C09104=1030.328,224.816,385.474,170.153,45.182,158.614
C09105=1030.334,225.065,385.447,170.156,45.180,158.614
C09106=1030.342,225.314,385.420,170.159,45.179,158.614
C09107=1030.349,225.562,385.392,170.162,45.178,158.614
C09108=1030.355,225.810,385.364,170.164,45.177,158.614
C09109=1030.361,226.059,385.337,170.167,45.176,158.614
C09110=1030.368,226.307,385.310,170.170,45.175,158.614
C09111=1030.375,226.555,385.283,170.173,45.174,158.614
C09112=1030.382,226.804,385.255,170.176,45.173,158.614
C09113=1030.388,227.052,385.227,170.180,45.172,158.614
C09114=1030.395,227.301,385.200,170.183,45.171,158.614
C09115=1030.402,227.549,385.173,170.186,45.170,158.614
C09116=1030.409,227.798,385.145,170.189,45.169,158.614
C09117=1030.416,228.046,385.118,170.192,45.168,158.615
C09118=1030.422,228.294,385.090,170.195,45.167,158.615
C09119=1030.428,228.543,385.062,170.198,45.166,158.615
C09120=1030.435,228.791,385.035,170.200,45.165,158.615
C09121=1030.442,229.039,385.007,170.203,45.164,158.615
C09122=1030.448,229.288,384.979,170.206,45.163,158.615
C09123=1030.455,229.536,384.952,170.209,45.162,158.615
C09124=1030.462,229.785,384.924,170.212,45.161,158.615
C09125=1030.468,230.033,384.896,170.215,45.160,158.615
C09126=1030.475,230.282,384.868,170.219,45.159,158.615
C09127=1030.482,230.530,384.841,170.222,45.158,158.616
C09128=1030.488,230.779,384.813,170.225,45.157,158.616
C09129=1030.495,231.027,384.785,170.228,45.157,158.616
C09130=1030.501,231.275,384.758,170.231,45.155,158.616
C09131=1030.507,231.523,384.729,170.234,45.155,158.616
C09132=1030.514,231.772,384.702,170.237,45.154,158.616
C09133=1030.521,232.020,384.674,170.240,45.153,158.616
C09134=1030.528,232.268,384.646,170.243,45.152,158.616
C09135=1030.534,232.517,384.618,170.246,45.151,158.616
C09136=1030.541,232.765,384.590,170.249,45.150,158.617
C09137=1030.547,233.014,384.562,170.252,45.149,158.617
C09138=1030.554,233.262,384.534,170.255,45.148,158.617
C09139=1030.560,233.511,384.506,170.258,45.148,158.617
C09140=1030.567,233.758,384.478,170.261,45.146,158.617
C09141=1030.576,234.068,384.443,170.265,45.145,158.617
C09142=1030.583,234.378,384.408,170.269,45.144,158.617
C09143=1030.591,234.686,384.374,170.273,45.143,158.617
C09144=1030.600,234.996,384.339,170.276,45.142,158.618
C09145=1030.607,235.243,384.311,170.280,45.141,158.618
C09146=1030.614,235.492,384.283,170.283,45.140,158.618
C09147=1030.619,235.741,384.255,170.286,45.139,158.618
C09148=1030.626,235.988,384.226,170.289,45.139,158.618
C09149=1030.633,236.237,384.198,170.292,45.138,158.618
C09150=1030.640,236.485,384.171,170.295,45.137,158.618
C09151=1030.647,236.734,384.143,170.298,45.136,158.619
C09152=1030.654,236.982,384.115,170.301,45.135,158.619
C09153=1030.659,237.230,384.086,170.305,45.134,158.619
C09154=1030.667,237.480,384.058,170.308,45.133,158.619
C09155=1030.674,237.727,384.030,170.311,45.132,158.619
C09156=1030.680,237.976,384.002,170.314,45.132,158.619
C09157=1030.687,238.224,383.973,170.317,45.131,158.619
C09158=1030.693,238.472,383.945,170.320,45.130,158.620
C09159=1030.700,238.721,383.917,170.324,45.129,158.620
C09160=1030.707,238.969,383.889,170.327,45.128,158.620
C09161=1030.713,239.217,383.861,170.330,45.128,158.620
C09162=1030.720,239.465,383.832,170.333,45.127,158.620
C09163=1030.727,239.714,383.805,170.336,45.126,158.620
C09164=1030.734,239.961,383.776,170.339,45.125,158.620
C09165=1030.740,240.211,383.747,170.343,45.124,158.620
C09166=1030.747,240.459,383.719,170.346,45.123,158.621
C09167=1030.753,240.707,383.691,170.349,45.123,158.621
C09168=1030.760,240.955,383.662,170.352,45.122,158.621
C09169=1030.766,241.204,383.634,170.355,45.121,158.621
C09170=1030.773,241.452,383.605,170.358,45.121,158.621
C09171=1030.779,241.700,383.576,170.361,45.120,158.621
C09172=1030.786,241.948,383.549,170.365,45.119,158.622
C09173=1030.793,242.197,383.519,170.368,45.118,158.622
C09174=1030.799,242.446,383.491,170.371,45.118,158.622
C09175=1030.806,242.694,383.462,170.374,45.117,158.622
C09176=1030.813,242.942,383.434,170.377,45.116,158.622
C09177=1030.819,243.190,383.406,170.380,45.115,158.622
C09178=1030.826,243.438,383.377,170.384,45.114,158.623
C09179=1030.832,243.686,383.348,170.387,45.113,158.623
C09180=1030.839,243.935,383.319,170.390,45.113,158.623
C09181=1030.847,244.242,383.284,170.394,45.112,158.623
C09182=1030.855,244.547,383.249,170.398,45.111,158.623
C09183=1030.863,244.854,383.214,170.402,45.111,158.624
C09184=1030.871,245.160,383.178,170.406,45.110,158.624
C09185=1030.877,245.409,383.149,170.410,45.109,158.624
C09186=1030.884,245.656,383.120,170.413,45.108,158.624
C09187=1030.891,245.905,383.091,170.416,45.108,158.624
C09188=1030.897,246.153,383.062,170.419,45.107,158.625
C09189=1030.903,246.402,383.033,170.422,45.106,158.625
C09190=1030.910,246.650,383.005,170.426,45.106,158.625
C09191=1030.916,246.898,382.976,170.429,45.105,158.625
C09192=1030.923,247.147,382.947,170.432,45.105,158.625
C09193=1030.929,247.395,382.918,170.435,45.104,158.626
C09194=1030.936,247.643,382.889,170.438,45.103,158.626
C09195=1030.943,247.891,382.860,170.442,45.103,158.626
C09196=1030.949,248.139,382.831,170.445,45.102,158.626
C09197=1030.959,248.501,382.789,170.449,45.101,158.626
C09198=1030.968,248.862,382.747,170.455,45.100,158.627
C09199=1030.978,249.224,382.704,170.460,45.099,158.627
C09200=1030.987,249.585,382.661,170.464,45.098,158.627
C09201=1030.994,249.832,382.633,170.468,45.098,158.627
C09202=1031.001,250.081,382.604,170.471,45.097,158.628
C09203=1031.007,250.329,382.575,170.474,45.097,158.628
C09204=1031.014,250.578,382.546,170.477,45.096,158.628
C09205=1031.020,250.826,382.516,170.481,45.095,158.628
C09206=1031.027,251.074,382.488,170.484,45.095,158.628
C09207=1031.034,251.322,382.459,170.487,45.094,158.629
C09208=1031.040,251.570,382.430,170.490,45.094,158.629
C09209=1031.047,251.819,382.399,170.493,45.093,158.629
C09210=1031.053,252.067,382.370,170.498,45.092,158.629
C09211=1031.060,252.315,382.342,170.501,45.092,158.629
C09212=1031.067,252.563,382.313,170.504,45.091,158.630
C09213=1031.073,252.812,382.284,170.507,45.091,158.630
C09214=1031.080,253.060,382.254,170.511,45.090,158.630
C09215=1031.087,253.308,382.224,170.514,45.089,158.630
C09216=1031.094,253.556,382.196,170.517,45.089,158.631
C09217=1031.101,253.805,382.167,170.521,45.088,158.631
C09218=1031.107,254.053,382.137,170.524,45.088,158.631
C09219=1031.113,254.300,382.108,170.527,45.087,158.631
C09220=1031.120,254.549,382.078,170.530,45.086,158.631
C09221=1031.127,254.797,382.049,170.535,45.086,158.632
C09222=1031.134,255.046,382.020,170.538,45.085,158.632
C09223=1031.141,255.293,381.991,170.541,45.085,158.632
C09224=1031.147,255.541,381.962,170.545,45.084,158.632
C09225=1031.154,255.790,381.932,170.548,45.084,158.633
C09226=1031.160,256.038,381.903,170.551,45.083,158.633
C09227=1031.168,256.286,381.874,170.554,45.082,158.633
C09228=1031.174,256.534,381.845,170.558,45.082,158.633
C09229=1031.181,256.783,381.815,170.562,45.082,158.633
C09230=1031.188,257.031,381.785,170.565,45.081,158.634
C09231=1031.194,257.280,381.756,170.569,45.080,158.634
C09232=1031.201,257.527,381.726,170.572,45.080,158.634
C09233=1031.209,257.776,381.698,170.575,45.079,158.634
C09234=1031.215,258.024,381.668,170.579,45.078,158.635
C09235=1031.222,258.272,381.638,170.582,45.078,158.635
C09236=1031.228,258.520,381.609,170.585,45.078,158.635
C09237=1031.235,258.768,381.579,170.589,45.077,158.635
C09238=1031.242,259.016,381.550,170.593,45.077,158.636
C09239=1031.250,259.264,381.521,170.596,45.076,158.636
C09240=1031.256,259.512,381.492,170.600,45.075,158.636
C09241=1031.263,259.761,381.461,170.603,45.075,158.636
C09242=1031.269,260.009,381.432,170.607,45.074,158.636
C09243=1031.276,260.257,381.402,170.610,45.073,158.637
C09244=1031.283,260.506,381.373,170.613,45.073,158.637
C09245=1031.290,260.753,381.343,170.617,45.073,158.637
C09246=1031.297,261.002,381.314,170.620,45.072,158.637
C09247=1031.304,261.249,381.285,170.624,45.072,158.638
C09248=1031.311,261.498,381.254,170.628,45.071,158.638
C09249=1031.317,261.746,381.225,170.631,45.071,158.638
C09250=1031.324,261.994,381.195,170.634,45.070,158.638
C09251=1031.330,262.242,381.165,170.638,45.070,158.639
C09252=1031.337,262.491,381.136,170.641,45.069,158.639
C09253=1031.347,262.850,381.091,170.647,45.069,158.639
C09254=1031.357,263.210,381.048,170.652,45.068,158.640
C09255=1031.366,263.570,381.005,170.657,45.068,158.640
C09256=1031.375,263.930,380.961,170.662,45.068,158.641
C09257=1031.382,264.178,380.931,170.666,45.067,158.641
C09258=1031.389,264.426,380.902,170.669,45.067,158.641
C09259=1031.396,264.674,380.871,170.672,45.067,158.641
C09260=1031.402,264.922,380.841,170.676,45.066,158.642
C09261=1031.409,265.170,380.811,170.680,45.066,158.642
C09262=1031.416,265.419,380.782,170.684,45.065,158.642
C09263=1031.423,265.667,380.751,170.687,45.065,158.642
C09264=1031.429,265.915,380.721,170.690,45.065,158.643
C09265=1031.436,266.163,380.691,170.694,45.064,158.643
C09266=1031.442,266.411,380.661,170.698,45.064,158.643
C09267=1031.450,266.659,380.631,170.702,45.063,158.644
C09268=1031.456,266.907,380.600,170.705,45.063,158.644
C09269=1031.463,267.155,380.571,170.708,45.063,158.644
C09270=1031.469,267.403,380.540,170.713,45.062,158.645
C09271=1031.476,267.652,380.510,170.716,45.062,158.645
C09272=1031.483,267.899,380.480,170.719,45.062,158.645
C09273=1031.489,268.148,380.449,170.723,45.061,158.645
C09274=1031.496,268.396,380.419,170.726,45.061,158.646
C09275=1031.503,268.643,380.389,170.731,45.060,158.646
C09276=1031.510,268.891,380.358,170.734,45.060,158.646
C09277=1031.517,269.139,380.328,170.737,45.060,158.647
C09278=1031.523,269.388,380.297,170.741,45.060,158.647
C09279=1031.530,269.635,380.267,170.744,45.059,158.647
C09280=1031.536,269.884,380.237,170.749,45.059,158.647
C09281=1031.543,270.132,380.207,170.752,45.059,158.648
C09282=1031.550,270.380,380.177,170.755,45.059,158.648
C09283=1031.557,270.628,380.145,170.759,45.058,158.648
C09284=1031.564,270.876,380.115,170.763,45.058,158.649
C09285=1031.570,271.124,380.085,170.767,45.058,158.649
C09286=1031.577,271.372,380.055,170.770,45.058,158.649
C09287=1031.583,271.620,380.023,170.775,45.058,158.650
C09288=1031.590,271.868,379.993,170.778,45.057,158.650
C09289=1031.597,272.116,379.963,170.781,45.057,158.650
C09290=1031.603,272.364,379.931,170.785,45.057,158.651
C09291=1031.610,272.612,379.901,170.788,45.056,158.651
C09292=1031.617,272.860,379.871,170.793,45.056,158.651
C09293=1031.624,273.108,379.840,170.796,45.056,158.652
C09294=1031.630,273.356,379.809,170.800,45.056,158.652
C09295=1031.636,273.604,379.779,170.804,45.056,158.652
C09296=1031.644,273.852,379.748,170.808,45.056,158.653
C09297=1031.650,274.100,379.717,170.811,45.056,158.653
C09298=1031.657,274.348,379.686,170.815,45.055,158.653
C09299=1031.663,274.596,379.656,170.819,45.055,158.654
C09300=1031.670,274.844,379.625,170.822,45.055,158.654
C09301=1031.677,275.092,379.594,170.826,45.055,158.654
C09302=1031.684,275.340,379.563,170.830,45.055,158.655
C09303=1031.691,275.588,379.532,170.834,45.055,158.655
C09304=1031.698,275.836,379.501,170.837,45.055,158.655
C09305=1031.704,276.085,379.471,170.842,45.054,158.656
C09306=1031.711,276.332,379.440,170.845,45.054,158.656
C09307=1031.718,276.580,379.410,170.849,45.054,158.656
C09308=1031.724,276.828,379.378,170.852,45.054,158.657
C09309=1031.734,277.192,379.332,170.858,45.053,158.657
C09310=1031.744,277.557,379.287,170.863,45.053,158.658
C09311=1031.754,277.921,379.242,170.870,45.053,158.658
C09312=1031.764,278.287,379.196,170.875,45.053,158.659
C09313=1031.771,278.534,379.165,170.879,45.053,158.659
C09314=1031.777,278.782,379.134,170.883,45.053,158.660
C09315=1031.784,279.030,379.102,170.886,45.053,158.660
C09316=1031.791,279.278,379.072,170.891,45.053,158.660
C09317=1031.797,279.526,379.040,170.894,45.053,158.661
C09318=1031.804,279.774,379.009,170.898,45.053,158.661
C09319=1031.811,280.022,378.977,170.902,45.052,158.661
C09320=1031.817,280.270,378.946,170.906,45.052,158.662
C09321=1031.824,280.518,378.915,170.909,45.053,158.662
C09322=1031.831,280.766,378.884,170.914,45.053,158.663
C09323=1031.837,281.014,378.852,170.917,45.052,158.663
C09324=1031.845,281.262,378.822,170.921,45.052,158.663
C09325=1031.852,281.510,378.790,170.925,45.053,158.664
C09326=1031.858,281.757,378.759,170.929,45.053,158.664
C09327=1031.865,282.005,378.727,170.932,45.052,158.664
C09328=1031.872,282.253,378.696,170.937,45.052,158.665
C09329=1031.878,282.501,378.664,170.940,45.052,158.665
C09330=1031.885,282.749,378.633,170.945,45.052,158.666
C09331=1031.892,282.997,378.602,170.948,45.052,158.666
C09332=1031.899,283.245,378.570,170.952,45.052,158.666
C09333=1031.905,283.493,378.539,170.956,45.053,158.667
C09334=1031.912,283.741,378.507,170.960,45.052,158.667
C09335=1031.919,283.989,378.476,170.964,45.052,158.668
C09336=1031.926,284.237,378.444,170.968,45.052,158.668
C09337=1031.932,284.484,378.413,170.972,45.052,158.669
C09338=1031.940,284.732,378.382,170.975,45.052,158.669
C09339=1031.946,284.980,378.351,170.980,45.052,158.669
C09340=1031.953,285.228,378.319,170.983,45.053,158.670
C09341=1031.960,285.476,378.288,170.988,45.052,158.670
C09342=1031.967,285.724,378.256,170.992,45.052,158.670
C09343=1031.974,285.972,378.225,170.995,45.053,158.671
C09344=1031.981,286.220,378.192,171.000,45.052,158.671
C09345=1031.988,286.467,378.161,171.003,45.053,158.672
C09346=1031.994,286.715,378.130,171.008,45.053,158.672
C09347=1032.000,286.964,378.098,171.012,45.052,158.673
C09348=1032.007,287.211,378.065,171.015,45.053,158.673
C09349=1032.014,287.459,378.034,171.020,45.053,158.673
C09350=1032.021,287.707,378.003,171.023,45.053,158.674
C09351=1032.028,287.955,377.970,171.028,45.053,158.674
C09352=1032.035,288.203,377.939,171.032,45.053,158.675
C09353=1032.042,288.450,377.907,171.035,45.053,158.675
C09354=1032.048,288.698,377.874,171.040,45.054,158.676
C09355=1032.055,288.946,377.843,171.043,45.054,158.676
C09356=1032.062,289.194,377.812,171.048,45.054,158.676
C09357=1032.069,289.441,377.779,171.052,45.054,158.677
C09358=1032.076,289.690,377.748,171.056,45.054,158.677
C09359=1032.082,289.937,377.715,171.060,45.055,158.678
C09360=1032.089,290.185,377.683,171.063,45.055,158.678
C09361=1032.096,290.432,377.651,171.068,45.055,158.679
C09362=1032.103,290.680,377.620,171.072,45.055,158.679
C09363=1032.110,290.929,377.587,171.076,45.055,158.680
C09364=1032.116,291.177,377.555,171.080,45.056,158.680
C09365=1032.124,291.441,377.521,171.085,45.055,158.680
C09366=1032.131,291.705,377.487,171.089,45.056,158.681
C09367=1032.139,291.969,377.453,171.094,45.056,158.682
C09368=1032.145,292.234,377.419,171.098,45.056,158.682
C09369=1032.153,292.482,377.386,171.102,45.056,158.682
C09370=1032.160,292.729,377.354,171.106,45.057,158.683
C09371=1032.166,292.978,377.322,171.111,45.056,158.683
C09372=1032.173,293.226,377.289,171.114,45.057,158.684
C09373=1032.180,293.473,377.257,171.119,45.057,158.684
C09374=1032.186,293.721,377.225,171.123,45.058,158.685
C09375=1032.193,293.968,377.193,171.127,45.057,158.685
C09376=1032.201,294.216,377.161,171.131,45.058,158.686
C09377=1032.207,294.464,377.128,171.136,45.058,158.686
C09378=1032.214,294.712,377.096,171.139,45.059,158.687
C09379=1032.221,294.960,377.063,171.144,45.059,158.687
C09380=1032.227,295.208,377.031,171.148,45.059,158.688
C09381=1032.234,295.455,376.998,171.152,45.059,158.688
C09382=1032.241,295.703,376.966,171.156,45.060,158.689
C09383=1032.248,295.951,376.933,171.161,45.060,158.689
C09384=1032.255,296.198,376.900,171.164,45.061,158.690
C09385=1032.261,296.446,376.868,171.169,45.061,158.690
C09386=1032.268,296.694,376.835,171.173,45.061,158.691
C09387=1032.274,296.942,376.802,171.177,45.062,158.691
C09388=1032.281,297.189,376.770,171.181,45.062,158.692
C09389=1032.288,297.437,376.737,171.186,45.063,158.692
C09390=1032.294,297.685,376.704,171.190,45.063,158.693
C09391=1032.301,297.932,376.672,171.194,45.063,158.693
C09392=1032.308,298.180,376.639,171.199,45.064,158.694
C09393=1032.317,298.540,376.591,171.205,45.064,158.695
C09394=1032.328,298.900,376.543,171.210,45.065,158.695
C09395=1032.337,299.260,376.496,171.217,45.066,158.696
C09396=1032.347,299.620,376.448,171.223,45.066,158.697
C09397=1032.354,299.867,376.415,171.228,45.067,158.698
C09398=1032.362,300.115,376.382,171.232,45.067,158.698
C09399=1032.368,300.363,376.349,171.236,45.068,158.699
C09400=1032.375,300.611,376.316,171.240,45.068,158.699
C09401=1032.381,300.858,376.283,171.245,45.068,158.700
C09402=1032.389,301.106,376.250,171.249,45.069,158.700
C09403=1032.395,301.353,376.217,171.253,45.069,158.701
C09404=1032.402,301.602,376.184,171.257,45.070,158.701
C09405=1032.409,301.849,376.152,171.262,45.070,158.702
C09406=1032.416,302.097,376.118,171.267,45.070,158.702
C09407=1032.423,302.344,376.086,171.270,45.071,158.703
C09408=1032.430,302.593,376.053,171.275,45.072,158.703
C09409=1032.437,302.839,376.020,171.279,45.072,158.704
C09410=1032.444,303.088,375.987,171.284,45.072,158.705
C09411=1032.450,303.335,375.953,171.289,45.073,158.705
C09412=1032.457,303.583,375.920,171.292,45.073,158.706
C09413=1032.464,303.830,375.888,171.297,45.074,158.706
C09414=1032.471,304.078,375.854,171.302,45.075,158.707
C09415=1032.478,304.326,375.821,171.306,45.075,158.707
C09416=1032.485,304.573,375.787,171.311,45.075,158.708
C09417=1032.493,304.821,375.755,171.314,45.076,158.708
C09418=1032.499,305.068,375.721,171.319,45.077,158.709
C09419=1032.506,305.316,375.688,171.324,45.077,158.710
C09420=1032.513,305.564,375.655,171.328,45.077,158.710
C09421=1032.525,305.957,375.602,171.335,45.079,158.711
C09422=1032.536,306.351,375.550,171.342,45.079,158.712
C09423=1032.547,306.744,375.496,171.349,45.080,158.713
C09424=1032.559,307.138,375.444,171.357,45.081,158.714
C09425=1032.565,307.386,375.411,171.361,45.082,158.714
C09426=1032.572,307.633,375.377,171.365,45.082,158.715
C09427=1032.579,307.881,375.343,171.370,45.083,158.716
C09428=1032.587,308.129,375.311,171.375,45.083,158.716
C09429=1032.594,308.376,375.277,171.379,45.084,158.717
C09430=1032.601,308.624,375.243,171.384,45.084,158.717
C09431=1032.608,308.871,375.210,171.389,45.085,158.718
C09432=1032.616,309.119,375.177,171.393,45.085,158.718
C09433=1032.622,309.366,375.144,171.398,45.086,158.719
C09434=1032.629,309.614,375.110,171.402,45.087,158.720
C09435=1032.637,309.862,375.076,171.406,45.088,158.720
C09436=1032.644,310.110,375.043,171.411,45.088,158.721
C09437=1032.651,310.357,375.010,171.416,45.088,158.721
C09438=1032.658,310.604,374.976,171.420,45.089,158.722
C09439=1032.665,310.852,374.942,171.425,45.089,158.723
C09440=1032.672,311.100,374.909,171.430,45.090,158.723
C09441=1032.680,311.347,374.875,171.434,45.091,158.724
C09442=1032.687,311.595,374.841,171.439,45.092,158.725
C09443=1032.693,311.842,374.807,171.444,45.092,158.725
C09444=1032.701,312.090,374.774,171.448,45.093,158.726
C09445=1032.707,312.338,374.739,171.453,45.094,158.727
C09446=1032.714,312.585,374.705,171.457,45.095,158.727
C09447=1032.721,312.833,374.670,171.462,45.095,158.728
C09448=1032.728,313.080,374.637,171.466,45.096,158.728
C09449=1032.735,313.327,374.603,171.471,45.097,158.729
C09450=1032.741,313.575,374.569,171.476,45.098,158.730
C09451=1032.749,313.823,374.535,171.481,45.098,158.730
C09452=1032.755,314.070,374.500,171.485,45.099,158.731
C09453=1032.763,314.318,374.466,171.490,45.100,158.732
C09454=1032.769,314.565,374.432,171.495,45.101,158.733
C09455=1032.776,314.813,374.398,171.500,45.102,158.733
C09456=1032.783,315.060,374.363,171.505,45.103,158.734
C09457=1032.790,315.308,374.330,171.508,45.104,158.734
C09458=1032.797,315.556,374.295,171.513,45.105,158.735
C09459=1032.804,315.803,374.261,171.518,45.106,158.736
C09460=1032.811,316.051,374.226,171.523,45.107,158.737
C09461=1032.818,316.298,374.192,171.528,45.107,158.737
C09462=1032.825,316.546,374.158,171.532,45.108,158.738
C09463=1032.832,316.794,374.123,171.537,45.109,158.739
C09464=1032.839,317.041,374.089,171.542,45.110,158.739
C09465=1032.846,317.289,374.054,171.547,45.111,158.740
C09466=1032.853,317.536,374.020,171.551,45.111,158.741
C09467=1032.860,317.784,373.985,171.556,45.112,158.741
C09468=1032.867,318.031,373.951,171.561,45.113,158.742
C09469=1032.875,318.278,373.917,171.566,45.114,158.743
C09470=1032.881,318.526,373.882,171.571,45.115,158.743
C09471=1032.889,318.773,373.848,171.576,45.116,158.744
C09472=1032.895,319.021,373.813,171.580,45.117,158.745
C09473=1032.903,319.268,373.778,171.585,45.118,158.746
C09474=1032.910,319.515,373.745,171.590,45.119,158.746
C09475=1032.917,319.763,373.709,171.595,45.120,158.747
C09476=1032.924,320.010,373.676,171.600,45.121,158.748
C09477=1032.935,320.409,373.619,171.608,45.122,158.749
C09478=1032.947,320.807,373.564,171.615,45.124,158.750
C09479=1032.958,321.206,373.507,171.624,45.125,158.751
C09480=1032.970,321.604,373.452,171.631,45.127,158.752
C09481=1032.977,321.852,373.417,171.637,45.128,158.753
C09482=1032.985,322.099,373.382,171.642,45.129,158.754
C09483=1032.992,322.347,373.348,171.647,45.130,158.755
C09484=1032.999,322.594,373.313,171.652,45.131,158.755
C09485=1033.006,322.841,373.279,171.656,45.132,158.756
C09486=1033.014,323.090,373.243,171.661,45.133,158.757
C09487=1033.021,323.337,373.209,171.666,45.134,158.758
C09488=1033.028,323.584,373.173,171.671,45.136,158.758
C09489=1033.036,323.831,373.139,171.676,45.136,158.759
C09490=1033.043,324.079,373.103,171.681,45.137,158.760
C09491=1033.050,324.327,373.070,171.687,45.138,158.761
C09492=1033.057,324.574,373.034,171.691,45.139,158.761
C09493=1033.065,324.822,373.000,171.697,45.140,158.762
C09494=1033.072,325.069,372.964,171.701,45.141,158.763
C09495=1033.079,325.316,372.930,171.706,45.142,158.764
C09496=1033.087,325.564,372.895,171.711,45.144,158.764
C09497=1033.094,325.811,372.860,171.716,45.145,158.765
C09498=1033.102,326.058,372.825,171.722,45.145,158.766
C09499=1033.109,326.306,372.789,171.727,45.147,158.767
C09500=1033.117,326.553,372.755,171.732,45.148,158.767
C09501=1033.124,326.801,372.719,171.737,45.149,158.768
C09502=1033.132,327.048,372.684,171.742,45.150,158.769
C09503=1033.139,327.295,372.649,171.748,45.151,158.770
C09504=1033.147,327.543,372.614,171.752,45.152,158.771
C09505=1033.153,327.791,372.579,171.757,45.153,158.771
C09506=1033.162,328.038,372.544,171.762,45.154,158.772
C09507=1033.169,328.285,372.509,171.767,45.156,158.773
C09508=1033.176,328.533,372.473,171.773,45.157,158.774
C09509=1033.183,328.780,372.437,171.778,45.158,158.775
C09510=1033.190,329.027,372.402,171.783,45.160,158.775
C09511=1033.197,329.275,372.367,171.788,45.161,158.776
C09512=1033.204,329.522,372.331,171.793,45.162,158.777
C09513=1033.212,329.770,372.296,171.798,45.163,158.778
C09514=1033.219,330.017,372.260,171.804,45.164,158.779
C09515=1033.227,330.265,372.224,171.809,45.166,158.780
C09516=1033.234,330.511,372.189,171.814,45.167,158.780
C09517=1033.241,330.759,372.153,171.819,45.168,158.781
C09518=1033.248,331.006,372.117,171.825,45.170,158.782
C09519=1033.256,331.254,372.082,171.830,45.171,158.783
C09520=1033.263,331.501,372.046,171.835,45.172,158.784
C09521=1033.270,331.748,372.010,171.840,45.173,158.785
C09522=1033.277,331.996,371.975,171.846,45.175,158.786
C09523=1033.285,332.243,371.938,171.851,45.176,158.786
C09524=1033.293,332.490,371.903,171.856,45.177,158.787
C09525=1033.300,332.738,371.868,171.861,45.179,158.788
C09526=1033.308,332.985,371.831,171.868,45.180,158.789
C09527=1033.315,333.232,371.796,171.873,45.181,158.790
C09528=1033.322,333.480,371.760,171.878,45.183,158.791
C09529=1033.329,333.727,371.724,171.883,45.185,158.792
C09530=1033.337,333.974,371.688,171.889,45.185,158.792
C09531=1033.345,334.222,371.652,171.894,45.187,158.793
C09532=1033.351,334.469,371.617,171.899,45.188,158.794
C09533=1033.364,334.863,371.559,171.908,45.191,158.796
C09534=1033.375,335.256,371.501,171.916,45.193,158.797
C09535=1033.387,335.651,371.444,171.925,45.195,158.798
C09536=1033.398,336.044,371.386,171.934,45.198,158.800
C09537=1033.406,336.292,371.350,171.939,45.199,158.801
C09538=1033.414,336.539,371.313,171.944,45.201,158.802
C09539=1033.421,336.787,371.277,171.950,45.202,158.803
C09540=1033.428,337.034,371.241,171.955,45.203,158.803
C09541=1033.435,337.281,371.205,171.961,45.205,158.804
C09542=1033.443,337.529,371.168,171.967,45.207,158.805
C09543=1033.451,337.775,371.131,171.972,45.208,158.806
C09544=1033.458,338.022,371.096,171.977,45.210,158.807
C09545=1033.465,338.270,371.059,171.983,45.211,158.808
C09546=1033.473,338.517,371.022,171.988,45.213,158.809
C09547=1033.480,338.765,370.986,171.994,45.214,158.810
C09548=1033.488,339.012,370.949,172.000,45.216,158.811
C09549=1033.495,339.258,370.913,172.005,45.217,158.812
C09550=1033.502,339.506,370.877,172.011,45.219,158.813
C09551=1033.510,339.754,370.840,172.016,45.221,158.814
C09552=1033.518,340.000,370.804,172.022,45.222,158.815
C09553=1033.526,340.248,370.767,172.027,45.224,158.816
C09554=1033.533,340.495,370.731,172.033,45.226,158.817
C09555=1033.541,340.743,370.694,172.039,45.227,158.818
C09556=1033.548,340.990,370.657,172.044,45.228,158.819
C09557=1033.556,341.236,370.621,172.050,45.230,158.820
C09558=1033.563,341.484,370.584,172.055,45.232,158.821
C09559=1033.571,341.731,370.547,172.061,45.234,158.822
C09560=1033.578,341.978,370.510,172.067,45.235,158.822
C09561=1033.586,342.225,370.473,172.072,45.237,158.824
C09562=1033.593,342.473,370.437,172.078,45.238,158.824
C09563=1033.600,342.720,370.400,172.084,45.241,158.826
C09564=1033.608,342.967,370.363,172.090,45.242,158.826
C09565=1033.615,343.214,370.326,172.095,45.244,158.828
C09566=1033.623,343.461,370.289,172.101,45.245,158.828
C09567=1033.631,343.708,370.251,172.106,45.247,158.830
C09568=1033.638,343.956,370.215,172.113,45.249,158.831
C09569=1033.646,344.203,370.178,172.118,45.251,158.831
C09570=1033.654,344.450,370.141,172.124,45.253,158.833
C09571=1033.661,344.697,370.103,172.130,45.255,158.834
C09572=1033.669,344.944,370.066,172.136,45.256,158.835
C09573=1033.676,345.191,370.029,172.141,45.258,158.836
C09574=1033.684,345.438,369.992,172.148,45.260,158.837
C09575=1033.691,345.685,369.955,172.153,45.261,158.838
C09576=1033.699,345.932,369.918,172.159,45.263,158.839
C09577=1033.707,346.180,369.880,172.164,45.265,158.840
C09578=1033.715,346.427,369.843,172.171,45.267,158.841
C09579=1033.722,346.674,369.806,172.176,45.269,158.842
C09580=1033.730,346.921,369.769,172.182,45.270,158.843
C09581=1033.737,347.168,369.731,172.188,45.273,158.844
C09582=1033.745,347.415,369.694,172.194,45.274,158.845
C09583=1033.752,347.662,369.657,172.200,45.276,158.846
C09584=1033.760,347.910,369.619,172.206,45.278,158.847
C09585=1033.768,348.157,369.582,172.212,45.280,158.848
C09586=1033.775,348.404,369.544,172.217,45.282,158.849
C09587=1033.783,348.651,369.507,172.224,45.284,158.850
C09588=1033.792,348.898,369.469,172.230,45.286,158.852
C09589=1033.803,349.289,369.409,172.239,45.289,158.853
C09590=1033.816,349.679,369.351,172.249,45.292,158.855
C09591=1033.828,350.070,369.291,172.258,45.295,158.857
C09592=1033.840,350.460,369.231,172.268,45.298,158.859
C09593=1033.847,350.707,369.193,172.273,45.300,158.860
C09594=1033.855,350.955,369.155,172.280,45.302,158.861
C09595=1033.863,351.201,369.117,172.286,45.304,158.862
C09596=1033.871,351.448,369.080,172.291,45.306,158.863
C09597=1033.879,351.695,369.042,172.298,45.309,158.864
C09598=1033.886,351.942,369.004,172.304,45.311,158.865
C09599=1033.894,352.189,368.966,172.310,45.313,158.866
C09600=1033.901,352.437,368.928,172.316,45.314,158.867
C09601=1033.910,352.683,368.890,172.323,45.317,158.869
C09602=1033.917,352.930,368.852,172.328,45.319,158.870
C09603=1033.925,353.177,368.814,172.335,45.321,158.871
C09604=1033.933,353.424,368.776,172.341,45.323,158.872
C09605=1033.940,353.672,368.738,172.347,45.325,158.873
C09606=1033.948,353.918,368.700,172.353,45.327,158.874
C09607=1033.957,354.165,368.662,172.360,45.330,158.876
C09608=1033.964,354.412,368.624,172.366,45.331,158.877
C09609=1033.972,354.660,368.586,172.372,45.334,158.878
C09610=1033.980,354.906,368.547,172.378,45.336,158.879
C09611=1033.988,355.153,368.509,172.385,45.338,158.880
C09612=1033.996,355.400,368.471,172.391,45.340,158.881
C09613=1034.004,355.647,368.433,172.397,45.343,158.883
C09614=1034.012,355.894,368.395,172.403,45.345,158.884
C09615=1034.020,356.141,368.356,172.410,45.347,158.885
C09616=1034.027,356.388,368.318,172.416,45.349,158.886
C09617=1034.036,356.635,368.280,172.423,45.351,158.888
C09618=1034.042,356.882,368.241,172.428,45.354,158.889
C09619=1034.051,357.129,368.202,172.435,45.356,158.890
C09620=1034.058,357.375,368.163,172.441,45.358,158.891
C09621=1034.067,357.622,368.125,172.448,45.361,158.892
C09622=1034.075,357.869,368.086,172.454,45.362,158.894
C09623=1034.082,358.116,368.048,172.460,45.365,158.895
C09624=1034.090,358.363,368.009,172.467,45.367,158.896
C09625=1034.099,358.610,367.971,172.473,45.370,158.897
C09626=1034.106,358.857,367.932,172.480,45.372,158.899
C09627=1034.115,359.103,367.893,172.486,45.374,158.900
C09628=1034.123,359.350,367.854,172.493,45.376,158.901
C09629=1034.130,359.597,367.816,172.500,45.379,158.902
C09630=1034.138,359.844,367.777,172.505,45.381,158.904
C09631=1034.147,360.091,367.738,172.512,45.384,158.905
C09632=1034.155,360.338,367.700,172.519,45.386,158.906
C09633=1034.163,360.584,367.661,172.525,45.389,158.907
C09634=1034.171,360.831,367.622,172.532,45.391,158.909
C09635=1034.178,361.079,367.583,172.539,45.394,158.910
C09636=1034.187,361.325,367.543,172.545,45.396,158.911
C09637=1034.194,361.572,367.505,172.552,45.398,158.913
C09638=1034.203,361.818,367.466,172.559,45.401,158.914
C09639=1034.211,362.065,367.426,172.565,45.403,158.915
C09640=1034.219,362.312,367.387,172.572,45.405,158.916
C09641=1034.227,362.558,367.348,172.579,45.408,158.918
C09642=1034.234,362.805,367.308,172.585,45.411,158.919
C09643=1034.242,363.052,367.270,172.591,45.414,158.920
C09644=1034.251,363.299,367.231,172.598,45.416,158.922
C09645=1034.263,363.696,367.167,172.609,45.420,158.924
C09646=1034.277,364.093,367.103,172.620,45.425,158.926
C09647=1034.289,364.489,367.040,172.630,45.429,158.928
C09648=1034.303,364.887,366.977,172.641,45.433,158.930
C09649=1034.310,365.133,366.938,172.649,45.435,158.932
C09650=1034.318,365.380,366.898,172.656,45.438,158.933
C09651=1034.327,365.626,366.859,172.663,45.440,158.935
C09652=1034.335,365.873,366.819,172.669,45.443,158.936
C09653=1034.343,366.120,366.780,172.676,45.446,158.937
C09654=1034.351,366.366,366.740,172.683,45.449,158.939
C09655=1034.359,366.613,366.700,172.690,45.451,158.940
C09656=1034.367,366.860,366.661,172.697,45.454,158.942
C09657=1034.376,367.107,366.621,172.703,45.456,158.943
C09658=1034.384,367.353,366.581,172.710,45.459,158.944
C09659=1034.393,367.600,366.541,172.717,45.462,158.946
C09660=1034.401,367.847,366.501,172.724,45.465,158.947
C09661=1034.409,368.093,366.462,172.731,45.468,158.949
C09662=1034.418,368.340,366.423,172.739,45.470,158.950
C09663=1034.426,368.586,366.382,172.745,45.473,158.951
C09664=1034.434,368.833,366.343,172.752,45.476,158.953
C09665=1034.442,369.080,366.302,172.759,45.479,158.954
C09666=1034.451,369.326,366.262,172.766,45.482,158.956
C09667=1034.460,369.573,366.223,172.773,45.484,158.957
C09668=1034.467,369.820,366.183,172.781,45.487,158.959
C09669=1034.475,370.066,366.143,172.788,45.490,158.960
C09670=1034.484,370.314,366.103,172.795,45.493,158.962
C09671=1034.492,370.560,366.062,172.802,45.495,158.963
C09672=1034.500,370.806,366.022,172.809,45.498,158.965
C09673=1034.509,371.053,365.982,172.817,45.501,158.966
C09674=1034.517,371.299,365.942,172.824,45.504,158.968
C09675=1034.526,371.546,365.901,172.831,45.507,158.969
C09676=1034.533,371.793,365.861,172.837,45.510,158.971
C09677=1034.542,372.039,365.821,172.845,45.514,158.972
C09678=1034.551,372.286,365.780,172.853,45.516,158.974
C09679=1034.559,372.532,365.739,172.860,45.519,158.975
C09680=1034.566,372.779,365.699,172.867,45.522,158.977
C09681=1034.575,373.025,365.659,172.874,45.525,158.978
C09682=1034.584,373.272,365.618,172.881,45.528,158.980
C09683=1034.592,373.518,365.577,172.889,45.531,158.981
C09684=1034.601,373.765,365.537,172.896,45.534,158.983
C09685=1034.609,374.011,365.496,172.904,45.537,158.984
C09686=1034.617,374.257,365.456,172.911,45.540,158.986
C09687=1034.626,374.504,365.415,172.918,45.543,158.987
C09688=1034.635,374.750,365.375,172.926,45.546,158.989
C09689=1034.643,374.997,365.334,172.933,45.550,158.991
C09690=1034.651,375.244,365.293,172.940,45.552,158.992
C09691=1034.660,375.491,365.252,172.948,45.556,158.994
C09692=1034.669,375.737,365.212,172.955,45.559,158.995
C09693=1034.677,375.984,365.171,172.962,45.562,158.997
C09694=1034.686,376.229,365.130,172.970,45.565,158.999
C09695=1034.694,376.476,365.089,172.978,45.568,159.000
C09696=1034.703,376.722,365.049,172.986,45.571,159.002
C09697=1034.712,376.969,365.008,172.993,45.575,159.003
C09698=1034.721,377.216,364.966,173.001,45.578,159.005
C09699=1034.729,377.462,364.925,173.008,45.581,159.007
C09700=1034.738,377.709,364.885,173.015,45.584,159.008
C09701=1034.745,377.918,364.850,173.022,45.587,159.010
C09702=1034.752,378.126,364.815,173.029,45.589,159.011
C09703=1034.760,378.335,364.780,173.035,45.593,159.012
C09704=1034.767,378.544,364.745,173.042,45.595,159.014
C09705=1034.774,378.751,364.710,173.049,45.598,159.015
C09706=1034.781,378.960,364.675,173.054,45.601,159.017
C09707=1034.788,379.170,364.640,173.061,45.603,159.018
C09708=1034.796,379.378,364.604,173.067,45.607,159.019
C09709=1034.804,379.624,364.564,173.075,45.610,159.021
C09710=1034.813,379.871,364.522,173.083,45.613,159.023
C09711=1034.822,380.117,364.480,173.091,45.616,159.025
C09712=1034.829,380.364,364.439,173.099,45.620,159.026
C09713=1034.838,380.610,364.397,173.106,45.623,159.028
C09714=1034.847,380.856,364.356,173.115,45.626,159.030
C09715=1034.856,381.103,364.314,173.122,45.630,159.031
C09716=1034.865,381.349,364.272,173.130,45.634,159.033
C09717=1034.873,381.595,364.231,173.138,45.637,159.035
C09718=1034.882,381.841,364.189,173.146,45.640,159.037
C09719=1034.891,382.088,364.147,173.154,45.644,159.038
C09720=1034.900,382.334,364.106,173.161,45.647,159.040
C09721=1034.909,382.580,364.064,173.170,45.651,159.042
C09722=1034.917,382.827,364.022,173.177,45.654,159.044
C09723=1034.926,383.073,363.980,173.185,45.658,159.045
C09724=1034.935,383.319,363.939,173.194,45.662,159.047
C09725=1034.944,383.565,363.897,173.201,45.665,159.049
C09726=1034.952,383.812,363.855,173.210,45.669,159.051
C09727=1034.961,384.058,363.813,173.218,45.672,159.052
C09728=1034.971,384.304,363.771,173.226,45.676,159.054
C09729=1034.980,384.550,363.729,173.234,45.679,159.056
C09730=1034.988,384.797,363.687,173.242,45.683,159.058
C09731=1034.997,385.043,363.645,173.251,45.686,159.060
C09732=1035.006,385.289,363.603,173.258,45.690,159.062
C09733=1035.015,385.535,363.561,173.266,45.694,159.063
C09734=1035.025,385.782,363.518,173.275,45.697,159.065
C09735=1035.034,386.028,363.477,173.284,45.701,159.067
C09736=1035.043,386.274,363.434,173.291,45.705,159.069
C09737=1035.052,386.520,363.392,173.299,45.708,159.071
C09738=1035.060,386.766,363.349,173.308,45.712,159.073
C09739=1035.069,387.013,363.308,173.317,45.716,159.074
C09740=1035.079,387.258,363.265,173.325,45.719,159.076
C09741=1035.088,387.506,363.223,173.333,45.723,159.078
C09742=1035.097,387.751,363.181,173.341,45.727,159.080
C09743=1035.106,387.997,363.138,173.349,45.731,159.082
C09744=1035.115,388.243,363.095,173.358,45.734,159.084
C09745=1035.124,388.489,363.052,173.367,45.738,159.086
C09746=1035.133,388.736,363.010,173.375,45.742,159.088
C09747=1035.142,388.982,362.968,173.384,45.746,159.090
C09748=1035.151,389.228,362.925,173.393,45.750,159.092
C09749=1035.160,389.474,362.882,173.401,45.754,159.093
C09750=1035.169,389.720,362.839,173.409,45.758,159.095
C09751=1035.178,389.966,362.797,173.417,45.762,159.097
C09752=1035.188,390.212,362.754,173.426,45.765,159.099
C09753=1035.197,390.459,362.711,173.435,45.770,159.101
C09754=1035.206,390.704,362.668,173.443,45.773,159.103
C09755=1035.215,390.951,362.624,173.452,45.778,159.105
C09756=1035.225,391.196,362.582,173.461,45.782,159.107
C09757=1035.233,391.442,362.539,173.469,45.785,159.109
C09758=1035.242,391.689,362.495,173.478,45.790,159.111
C09759=1035.252,391.934,362.452,173.487,45.793,159.113
C09760=1035.261,392.181,362.409,173.495,45.798,159.115
C09761=1035.270,392.407,362.370,173.504,45.801,159.117
C09762=1035.278,392.633,362.329,173.512,45.805,159.119
C09763=1035.286,392.858,362.290,173.520,45.809,159.121
C09764=1035.295,393.085,362.250,173.528,45.812,159.123
C09765=1035.304,393.311,362.210,173.536,45.816,159.125
C09766=1035.312,393.537,362.171,173.545,45.820,159.126
C09767=1035.321,393.763,362.130,173.552,45.824,159.128
C09768=1035.329,393.990,362.090,173.561,45.828,159.130
C09769=1035.339,394.235,362.047,173.570,45.832,159.132
C09770=1035.348,394.481,362.004,173.578,45.836,159.134
C09771=1035.357,394.728,361.960,173.587,45.841,159.137
C09772=1035.367,394.973,361.916,173.597,45.845,159.139
C09773=1035.376,395.219,361.873,173.606,45.849,159.141
C09774=1035.385,395.466,361.829,173.615,45.853,159.143
C09775=1035.394,395.711,361.785,173.624,45.858,159.145
C09776=1035.404,395.957,361.742,173.633,45.862,159.147
C09777=1035.414,396.203,361.698,173.643,45.866,159.149
C09778=1035.423,396.448,361.654,173.651,45.870,159.151
C09779=1035.432,396.695,361.610,173.660,45.874,159.153
C09780=1035.442,396.940,361.566,173.669,45.879,159.156
C09781=1035.451,397.187,361.522,173.679,45.883,159.158
C09782=1035.461,397.433,361.478,173.688,45.888,159.160
C09783=1035.470,397.677,361.434,173.697,45.892,159.162
C09784=1035.480,397.923,361.390,173.707,45.896,159.165
C09785=1035.490,398.169,361.346,173.716,45.901,159.167
C09786=1035.499,398.416,361.302,173.725,45.906,159.169
C09787=1035.508,398.662,361.258,173.735,45.910,159.171
C09788=1035.519,398.907,361.213,173.744,45.914,159.173
C09789=1035.528,399.153,361.169,173.753,45.919,159.175
C09790=1035.538,399.399,361.125,173.763,45.923,159.178
C09791=1035.547,399.645,361.080,173.772,45.927,159.180
C09792=1035.557,399.891,361.036,173.782,45.932,159.182
C09793=1035.566,400.136,360.992,173.792,45.937,159.185
C09794=1035.576,400.382,360.947,173.801,45.941,159.187
C09795=1035.586,400.628,360.903,173.811,45.946,159.189
C09796=1035.595,400.874,360.858,173.820,45.950,159.191
C09797=1035.605,401.120,360.814,173.830,45.955,159.194
C09798=1035.614,401.365,360.769,173.839,45.960,159.196
C09799=1035.624,401.611,360.724,173.849,45.964,159.198
C09800=1035.634,401.856,360.679,173.859,45.969,159.201
C09801=1035.644,402.102,360.634,173.869,45.974,159.203
C09802=1035.654,402.349,360.590,173.878,45.979,159.205
C09803=1035.663,402.594,360.545,173.888,45.983,159.208
C09804=1035.673,402.840,360.500,173.897,45.988,159.210
C09805=1035.683,403.085,360.455,173.908,45.992,159.212
C09806=1035.692,403.331,360.411,173.918,45.998,159.215
C09807=1035.703,403.577,360.365,173.927,46.002,159.217
C09808=1035.713,403.822,360.320,173.937,46.007,159.220
C09809=1035.722,404.068,360.274,173.947,46.012,159.222
C09810=1035.732,404.313,360.230,173.957,46.017,159.224
C09811=1035.742,404.559,360.184,173.968,46.022,159.227
C09812=1035.752,404.804,360.139,173.977,46.027,159.229
C09813=1035.761,405.051,360.093,173.987,46.032,159.232
C09814=1035.771,405.296,360.048,173.998,46.036,159.234
C09815=1035.781,405.541,360.003,174.008,46.041,159.237
C09816=1035.791,405.787,359.958,174.017,46.046,159.239
C09817=1035.801,406.033,359.913,174.028,46.051,159.242
C09818=1035.811,406.279,359.866,174.038,46.056,159.244
C09819=1035.821,406.524,359.821,174.049,46.061,159.247
C09820=1035.831,406.770,359.775,174.058,46.066,159.249
C09821=1035.841,407.006,359.731,174.068,46.071,159.252
C09822=1035.851,407.242,359.688,174.079,46.076,159.254
C09823=1035.860,407.479,359.644,174.088,46.081,159.257
C09824=1035.870,407.714,359.600,174.098,46.085,159.259
C09825=1035.880,407.951,359.556,174.108,46.091,159.261
C09826=1035.890,408.187,359.512,174.118,46.095,159.264
C09827=1035.899,408.423,359.468,174.129,46.100,159.266
C09828=1035.910,408.660,359.424,174.138,46.106,159.269
C09829=1035.919,408.905,359.378,174.149,46.111,159.271
C09830=1035.930,409.150,359.332,174.159,46.116,159.274
C09831=1035.940,409.396,359.286,174.170,46.121,159.277
C09832=1035.951,409.642,359.240,174.181,46.126,159.279
C09833=1035.960,409.887,359.194,174.191,46.131,159.282
C09834=1035.971,410.132,359.148,174.202,46.136,159.284
C09835=1035.981,410.378,359.102,174.212,46.142,159.287
C09836=1035.992,410.624,359.056,174.223,46.147,159.290
C09837=1036.002,410.869,359.009,174.234,46.152,159.292
C09838=1036.013,411.115,358.964,174.245,46.157,159.295
C09839=1036.024,411.360,358.917,174.256,46.163,159.298
C09840=1036.033,411.606,358.870,174.267,46.168,159.301
C09841=1036.044,411.851,358.823,174.277,46.173,159.303
C09842=1036.054,412.097,358.777,174.288,46.179,159.306
C09843=1036.064,412.342,358.730,174.299,46.184,159.309
C09844=1036.075,412.588,358.684,174.310,46.190,159.311
C09845=1036.085,412.833,358.637,174.322,46.195,159.314
C09846=1036.096,413.079,358.591,174.333,46.201,159.317
C09847=1036.106,413.324,358.544,174.344,46.206,159.320
C09848=1036.116,413.569,358.497,174.354,46.212,159.323
C09849=1036.127,413.814,358.450,174.366,46.217,159.325
C09850=1036.137,414.060,358.404,174.377,46.223,159.328
C09851=1036.148,414.305,358.357,174.388,46.228,159.331
C09852=1036.159,414.551,358.309,174.399,46.234,159.334
C09853=1036.169,414.796,358.262,174.411,46.240,159.337
C09854=1036.180,415.041,358.215,174.422,46.245,159.339
C09855=1036.190,415.286,358.168,174.434,46.251,159.342
C09856=1036.202,415.532,358.121,174.445,46.257,159.345
C09857=1036.212,415.777,358.074,174.456,46.263,159.348
C09858=1036.222,416.023,358.027,174.468,46.268,159.351
C09859=1036.234,416.268,357.979,174.479,46.274,159.354
C09860=1036.244,416.513,357.932,174.491,46.279,159.357
C09861=1036.255,416.758,357.885,174.502,46.285,159.360
C09862=1036.266,417.004,357.838,174.514,46.291,159.363
C09863=1036.277,417.249,357.789,174.525,46.297,159.366
C09864=1036.288,417.494,357.743,174.537,46.302,159.369
C09865=1036.298,417.739,357.695,174.549,46.308,159.372
C09866=1036.309,417.985,357.647,174.561,46.314,159.375
C09867=1036.320,418.230,357.599,174.573,46.320,159.378
C09868=1036.330,418.476,357.552,174.584,46.326,159.381
C09869=1036.341,418.720,357.504,174.596,46.332,159.384
C09870=1036.352,418.966,357.456,174.609,46.338,159.387
C09871=1036.364,419.211,357.408,174.620,46.344,159.390
C09872=1036.374,419.456,357.361,174.632,46.350,159.393
C09873=1036.385,419.701,357.312,174.644,46.356,159.396
C09874=1036.396,419.946,357.264,174.656,46.362,159.399
C09875=1036.407,420.191,357.216,174.668,46.368,159.402
C09876=1036.418,420.437,357.168,174.680,46.374,159.405
C09877=1036.429,420.682,357.120,174.693,46.380,159.408
C09878=1036.439,420.927,357.072,174.705,46.386,159.412
C09879=1036.451,421.172,357.024,174.717,46.392,159.415
C09880=1036.463,421.417,356.975,174.729,46.399,159.418
C09881=1036.473,421.657,356.928,174.741,46.405,159.421
C09882=1036.484,421.899,356.880,174.754,46.411,159.424
C09883=1036.495,422.139,356.832,174.766,46.417,159.427
C09884=1036.506,422.380,356.785,174.778,46.423,159.430
C09885=1036.518,422.620,356.737,174.790,46.429,159.434
C09886=1036.528,422.861,356.690,174.802,46.435,159.437
C09887=1036.540,423.101,356.642,174.815,46.441,159.440
C09888=1036.551,423.342,356.594,174.827,46.448,159.443
C09889=1036.562,423.587,356.545,174.840,46.454,159.446
C09890=1036.573,423.832,356.497,174.852,46.460,159.450
C09891=1036.585,424.077,356.448,174.865,46.467,159.453
C09892=1036.596,424.322,356.399,174.879,46.473,159.456
C09893=1036.607,424.567,356.350,174.891,46.480,159.460
C09894=1036.618,424.812,356.300,174.904,46.486,159.463
C09895=1036.630,425.056,356.251,174.917,46.492,159.466
C09896=1036.641,425.301,356.202,174.929,46.499,159.470
C09897=1036.653,425.547,356.153,174.943,46.505,159.473
C09898=1036.665,425.791,356.104,174.956,46.512,159.477
C09899=1036.676,426.036,356.055,174.969,46.518,159.480
C09900=1036.687,426.281,356.005,174.981,46.525,159.483
C09901=1036.699,426.527,355.956,174.995,46.531,159.487
C09902=1036.710,426.771,355.906,175.008,46.538,159.490
C09903=1036.722,427.015,355.857,175.021,46.545,159.494
C09904=1036.734,427.261,355.808,175.035,46.551,159.497
C09905=1036.745,427.505,355.758,175.048,46.558,159.501
C09906=1036.758,427.750,355.709,175.062,46.565,159.504
C09907=1036.768,427.995,355.659,175.075,46.572,159.508
C09908=1036.780,428.240,355.610,175.089,46.578,159.511
C09909=1036.792,428.484,355.559,175.102,46.585,159.515
C09910=1036.803,428.729,355.509,175.116,46.592,159.518
C09911=1036.815,428.974,355.460,175.129,46.599,159.522
C09912=1036.826,429.219,355.409,175.143,46.605,159.526
C09913=1036.838,429.464,355.359,175.157,46.612,159.529
C09914=1036.851,429.708,355.309,175.170,46.619,159.533
C09915=1036.862,429.953,355.259,175.184,46.626,159.537
C09916=1036.874,430.198,355.209,175.198,46.633,159.540
C09917=1036.886,430.442,355.159,175.212,46.640,159.544
C09918=1036.897,430.687,355.108,175.226,46.647,159.547
C09919=1036.910,430.931,355.058,175.240,46.654,159.551
C09920=1036.922,431.176,355.007,175.254,46.661,159.555
C09921=1036.933,431.420,354.957,175.269,46.668,159.559
C09922=1036.946,431.665,354.907,175.282,46.675,159.562
C09923=1036.957,431.910,354.856,175.296,46.682,159.566
C09924=1036.970,432.154,354.806,175.311,46.690,159.570
C09925=1036.982,432.399,354.755,175.325,46.697,159.574
C09926=1036.994,432.644,354.704,175.339,46.703,159.578
C09927=1037.007,432.888,354.653,175.354,46.711,159.581
C09928=1037.019,433.132,354.602,175.368,46.718,159.585
C09929=1037.031,433.377,354.552,175.382,46.725,159.589
C09930=1037.043,433.622,354.501,175.397,46.732,159.593
C09931=1037.055,433.866,354.449,175.413,46.740,159.597
C09932=1037.068,434.110,354.399,175.427,46.747,159.601
C09933=1037.081,434.354,354.348,175.442,46.754,159.605
C09934=1037.092,434.600,354.297,175.456,46.762,159.609
C09935=1037.106,434.844,354.245,175.471,46.769,159.613
C09936=1037.117,435.088,354.194,175.486,46.776,159.617
C09937=1037.130,435.333,354.143,175.501,46.783,159.621
C09938=1037.142,435.577,354.092,175.516,46.791,159.625
C09939=1037.154,435.822,354.040,175.530,46.799,159.629
C09940=1037.167,436.066,353.988,175.546,46.806,159.633
C09941=1037.187,436.456,353.906,175.570,46.818,159.639
C09942=1037.207,436.847,353.824,175.595,46.830,159.646
C09943=1037.227,437.237,353.741,175.619,46.842,159.652
C09944=1037.247,437.628,353.658,175.643,46.854,159.659
C09945=1037.265,437.967,353.586,175.666,46.865,159.665
C09946=1037.283,438.306,353.513,175.687,46.876,159.671
C09947=1037.300,438.645,353.441,175.709,46.886,159.676
C09948=1037.318,438.984,353.368,175.731,46.897,159.682
C09949=1037.330,439.228,353.316,175.747,46.905,159.687
C09950=1037.344,439.472,353.264,175.763,46.913,159.691
C09951=1037.357,439.717,353.211,175.778,46.921,159.695
C09952=1037.369,439.960,353.159,175.794,46.929,159.700
C09953=1037.383,440.204,353.107,175.810,46.937,159.704
C09954=1037.396,440.449,353.054,175.827,46.945,159.708
C09955=1037.409,440.693,353.001,175.843,46.953,159.713
C09956=1037.422,440.937,352.948,175.859,46.961,159.717
C09957=1037.434,441.181,352.896,175.875,46.969,159.722
C09958=1037.447,441.425,352.843,175.892,46.977,159.726
C09959=1037.461,441.669,352.790,175.908,46.985,159.730
C09960=1037.474,441.913,352.737,175.924,46.993,159.735
C09961=1037.487,442.157,352.684,175.941,47.001,159.739
C09962=1037.500,442.401,352.631,175.958,47.009,159.744
C09963=1037.513,442.645,352.578,175.975,47.017,159.749
C09964=1037.527,442.889,352.525,175.991,47.025,159.753
C09965=1037.540,443.133,352.472,176.008,47.034,159.758
C09966=1037.554,443.377,352.418,176.025,47.042,159.762
C09967=1037.567,443.621,352.365,176.042,47.050,159.767
C09968=1037.580,443.865,352.311,176.060,47.058,159.772
C09969=1037.594,444.107,352.258,176.076,47.066,159.776
C09970=1037.608,444.350,352.205,176.093,47.075,159.781
C09971=1037.622,444.594,352.152,176.110,47.083,159.785
C09972=1037.637,444.838,352.100,176.128,47.091,159.790
C09973=1037.651,445.081,352.048,176.145,47.099,159.795
C09974=1037.667,445.324,351.997,176.162,47.107,159.799
C09975=1037.683,445.567,351.945,176.179,47.115,159.804
C09976=1037.700,445.812,351.895,176.197,47.123,159.808
C09977=1037.718,446.055,351.845,176.215,47.130,159.813
C09978=1037.735,446.299,351.795,176.233,47.138,159.817
C09979=1037.754,446.543,351.746,176.251,47.145,159.822
C09980=1037.773,446.787,351.697,176.269,47.153,159.827
C09981=1037.793,447.032,351.649,176.287,47.160,159.831
C09982=1037.814,447.275,351.601,176.305,47.167,159.836
C09983=1037.834,447.520,351.553,176.322,47.174,159.840
C09984=1037.855,447.765,351.506,176.341,47.181,159.845
C09985=1037.877,448.009,351.459,176.360,47.188,159.849
C09986=1037.899,448.254,351.414,176.378,47.194,159.853
C09987=1037.922,448.499,351.368,176.396,47.201,159.858
C09988=1037.946,448.744,351.323,176.415,47.208,159.862
C09989=1037.970,448.988,351.278,176.433,47.215,159.867
C09990=1037.995,449.233,351.233,176.452,47.221,159.871
C09991=1038.019,449.478,351.190,176.471,47.227,159.875
C09992=1038.045,449.724,351.146,176.489,47.233,159.880
C09993=1038.072,449.969,351.104,176.509,47.240,159.884
C09994=1038.099,450.214,351.061,176.529,47.246,159.889
C09995=1038.127,450.459,351.019,176.547,47.252,159.893
C09996=1038.154,450.704,350.977,176.566,47.258,159.897
//INST
///DATE 2021/06/25 14:49
///ATTR SC,RW,RJ
////FRAME ROBOT
///GROUP1 RB1
NOP
MOVL C00000 V=800.0 PL=0
MOVL C00001 V=800.0 PL=0
MOVL C00002 V=800.0 PL=0
MOVL C00003 V=800.0 PL=0
MOVL C00004 V=800.0 PL=0
MOVL C00005 V=800.0 PL=0
MOVL C00006 V=800.0 PL=0
MOVL C00007 V=800.0 PL=0
MOVL C00008 V=800.0 PL=0
MOVL C00009 V=800.0 PL=0
MOVL C00010 V=800.0 PL=0
MOVL C00011 V=800.0 PL=0
MOVL C00012 V=800.0 PL=0
MOVL C00013 V=800.0 PL=0
MOVL C00014 V=800.0 PL=0
MOVL C00015 V=800.0 PL=0
MOVL C00016 V=800.0 PL=0
MOVL C00017 V=800.0 PL=0
MOVL C00018 V=800.0 PL=0
MOVL C00019 V=800.0 PL=0
MOVL C00020 V=800.0 PL=0
MOVL C00021 V=800.0 PL=0
MOVL C00022 V=800.0 PL=0
MOVL C00023 V=800.0 PL=0
MOVL C00024 V=800.0 PL=0
MOVL C00025 V=800.0 PL=0
MOVL C00026 V=800.0 PL=0
MOVL C00027 V=800.0 PL=0
MOVL C00028 V=800.0 PL=0
MOVL C00029 V=800.0 PL=0
MOVL C00030 V=800.0 PL=0
MOVL C00031 V=800.0 PL=0
MOVL C00032 V=800.0 PL=0
MOVL C00033 V=800.0 PL=0
MOVL C00034 V=800.0 PL=0
MOVL C00035 V=800.0 PL=0
MOVL C00036 V=800.0 PL=0
MOVL C00037 V=800.0 PL=0
MOVL C00038 V=800.0 PL=0
MOVL C00039 V=800.0 PL=0
MOVL C00040 V=800.0 PL=0
MOVL C00041 V=800.0 PL=0
MOVL C00042 V=800.0 PL=0
MOVL C00043 V=800.0 PL=0
MOVL C00044 V=800.0 PL=0
MOVL C00045 V=800.0 PL=0
MOVL C00046 V=800.0 PL=0
MOVL C00047 V=800.0 PL=0
MOVL C00048 V=800.0 PL=0
MOVL C00049 V=800.0 PL=0
MOVL C00050 V=800.0 PL=0
MOVL C00051 V=800.0 PL=0
MOVL C00052 V=800.0 PL=0
MOVL C00053 V=800.0 PL=0
MOVL C00054 V=800.0 PL=0
MOVL C00055 V=800.0 PL=0
MOVL C00056 V=800.0 PL=0
MOVL C00057 V=800.0 PL=0
MOVL C00058 V=800.0 PL=0
MOVL C00059 V=800.0 PL=0
MOVL C00060 V=800.0 PL=0
MOVL C00061 V=800.0 PL=0
MOVL C00062 V=800.0 PL=0
MOVL C00063 V=800.0 PL=0
MOVL C00064 V=800.0 PL=0
MOVL C00065 V=800.0 PL=0
MOVL C00066 V=800.0 PL=0
MOVL C00067 V=800.0 PL=0
MOVL C00068 V=800.0 PL=0
MOVL C00069 V=800.0 PL=0
MOVL C00070 V=800.0 PL=0
MOVL C00071 V=800.0 PL=0
MOVL C00072 V=800.0 PL=0
MOVL C00073 V=800.0 PL=0
MOVL C00074 V=800.0 PL=0
MOVL C00075 V=800.0 PL=0
MOVL C00076 V=800.0 PL=0
MOVL C00077 V=800.0 PL=0
MOVL C00078 V=800.0 PL=0
MOVL C00079 V=800.0 PL=0
MOVL C00080 V=800.0 PL=0
MOVL C00081 V=800.0 PL=0
MOVL C00082 V=800.0 PL=0
MOVL C00083 V=800.0 PL=0
MOVL C00084 V=800.0 PL=0
MOVL C00085 V=800.0 PL=0
MOVL C00086 V=800.0 PL=0
MOVL C00087 V=800.0 PL=0
MOVL C00088 V=800.0 PL=0
MOVL C00089 V=800.0 PL=0
MOVL C00090 V=800.0 PL=0
MOVL C00091 V=800.0 PL=0
MOVL C00092 V=800.0 PL=0
MOVL C00093 V=800.0 PL=0
MOVL C00094 V=800.0 PL=0
MOVL C00095 V=800.0 PL=0
MOVL C00096 V=800.0 PL=0
MOVL C00097 V=800.0 PL=0
MOVL C00098 V=800.0 PL=0
MOVL C00099 V=800.0 PL=0
MOVL C00100 V=800.0 PL=0
MOVL C00101 V=800.0 PL=0
MOVL C00102 V=800.0 PL=0
MOVL C00103 V=800.0 PL=0
MOVL C00104 V=800.0 PL=0
MOVL C00105 V=800.0 PL=0
MOVL C00106 V=800.0 PL=0
MOVL C00107 V=800.0 PL=0
MOVL C00108 V=800.0 PL=0
MOVL C00109 V=800.0 PL=0
MOVL C00110 V=800.0 PL=0
MOVL C00111 V=800.0 PL=0
MOVL C00112 V=800.0 PL=0
MOVL C00113 V=800.0 PL=0
MOVL C00114 V=800.0 PL=0
MOVL C00115 V=800.0 PL=0
MOVL C00116 V=800.0 PL=0
MOVL C00117 V=800.0 PL=0
MOVL C00118 V=800.0 PL=0
MOVL C00119 V=800.0 PL=0
MOVL C00120 V=800.0 PL=0
MOVL C00121 V=800.0 PL=0
MOVL C00122 V=800.0 PL=0
MOVL C00123 V=800.0 PL=0
MOVL C00124 V=800.0 PL=0
MOVL C00125 V=800.0 PL=0
MOVL C00126 V=800.0 PL=0
MOVL C00127 V=800.0 PL=0
MOVL C00128 V=800.0 PL=0
MOVL C00129 V=800.0 PL=0
MOVL C00130 V=800.0 PL=0
MOVL C00131 V=800.0 PL=0
MOVL C00132 V=800.0 PL=0
MOVL C00133 V=800.0 PL=0
MOVL C00134 V=800.0 PL=0
MOVL C00135 V=800.0 PL=0
MOVL C00136 V=800.0 PL=0
MOVL C00137 V=800.0 PL=0
MOVL C00138 V=800.0 PL=0
MOVL C00139 V=800.0 PL=0
MOVL C00140 V=800.0 PL=0
MOVL C00141 V=800.0 PL=0
MOVL C00142 V=800.0 PL=0
MOVL C00143 V=800.0 PL=0
MOVL C00144 V=800.0 PL=0
MOVL C00145 V=800.0 PL=0
MOVL C00146 V=800.0 PL=0
MOVL C00147 V=800.0 PL=0
MOVL C00148 V=800.0 PL=0
MOVL C00149 V=800.0 PL=0
MOVL C00150 V=800.0 PL=0
MOVL C00151 V=800.0 PL=0
MOVL C00152 V=800.0 PL=0
MOVL C00153 V=800.0 PL=0
MOVL C00154 V=800.0 PL=0
MOVL C00155 V=800.0 PL=0
MOVL C00156 V=800.0 PL=0
MOVL C00157 V=800.0 PL=0
MOVL C00158 V=800.0 PL=0
MOVL C00159 V=800.0 PL=0
MOVL C00160 V=800.0 PL=0
MOVL C00161 V=800.0 PL=0
MOVL C00162 V=800.0 PL=0
MOVL C00163 V=800.0 PL=0
MOVL C00164 V=800.0 PL=0
MOVL C00165 V=800.0 PL=0
MOVL C00166 V=800.0 PL=0
MOVL C00167 V=800.0 PL=0
MOVL C00168 V=800.0 PL=0
MOVL C00169 V=800.0 PL=0
MOVL C00170 V=800.0 PL=0
MOVL C00171 V=800.0 PL=0
MOVL C00172 V=800.0 PL=0
MOVL C00173 V=800.0 PL=0
MOVL C00174 V=800.0 PL=0
MOVL C00175 V=800.0 PL=0
MOVL C00176 V=800.0 PL=0
MOVL C00177 V=800.0 PL=0
MOVL C00178 V=800.0 PL=0
MOVL C00179 V=800.0 PL=0
MOVL C00180 V=800.0 PL=0
MOVL C00181 V=800.0 PL=0
MOVL C00182 V=800.0 PL=0
MOVL C00183 V=800.0 PL=0
MOVL C00184 V=800.0 PL=0
MOVL C00185 V=800.0 PL=0
MOVL C00186 V=800.0 PL=0
MOVL C00187 V=800.0 PL=0
MOVL C00188 V=800.0 PL=0
MOVL C00189 V=800.0 PL=0
MOVL C00190 V=800.0 PL=0
MOVL C00191 V=800.0 PL=0
MOVL C00192 V=800.0 PL=0
MOVL C00193 V=800.0 PL=0
MOVL C00194 V=800.0 PL=0
MOVL C00195 V=800.0 PL=0
MOVL C00196 V=800.0 PL=0
MOVL C00197 V=800.0 PL=0
MOVL C00198 V=800.0 PL=0
MOVL C00199 V=800.0 PL=0
MOVL C00200 V=800.0 PL=0
MOVL C00201 V=800.0 PL=0
MOVL C00202 V=800.0 PL=0
MOVL C00203 V=800.0 PL=0
MOVL C00204 V=800.0 PL=0
MOVL C00205 V=800.0 PL=0
MOVL C00206 V=800.0 PL=0
MOVL C00207 V=800.0 PL=0
MOVL C00208 V=800.0 PL=0
MOVL C00209 V=800.0 PL=0
MOVL C00210 V=800.0 PL=0
MOVL C00211 V=800.0 PL=0
MOVL C00212 V=800.0 PL=0
MOVL C00213 V=800.0 PL=0
MOVL C00214 V=800.0 PL=0
MOVL C00215 V=800.0 PL=0
MOVL C00216 V=800.0 PL=0
MOVL C00217 V=800.0 PL=0
MOVL C00218 V=800.0 PL=0
MOVL C00219 V=800.0 PL=0
MOVL C00220 V=800.0 PL=0
MOVL C00221 V=800.0 PL=0
MOVL C00222 V=800.0 PL=0
MOVL C00223 V=800.0 PL=0
MOVL C00224 V=800.0 PL=0
MOVL C00225 V=800.0 PL=0
MOVL C00226 V=800.0 PL=0
MOVL C00227 V=800.0 PL=0
MOVL C00228 V=800.0 PL=0
MOVL C00229 V=800.0 PL=0
MOVL C00230 V=800.0 PL=0
MOVL C00231 V=800.0 PL=0
MOVL C00232 V=800.0 PL=0
MOVL C00233 V=800.0 PL=0
MOVL C00234 V=800.0 PL=0
MOVL C00235 V=800.0 PL=0
MOVL C00236 V=800.0 PL=0
MOVL C00237 V=800.0 PL=0
MOVL C00238 V=800.0 PL=0
MOVL C00239 V=800.0 PL=0
MOVL C00240 V=800.0 PL=0
MOVL C00241 V=800.0 PL=0
MOVL C00242 V=800.0 PL=0
MOVL C00243 V=800.0 PL=0
MOVL C00244 V=800.0 PL=0
MOVL C00245 V=800.0 PL=0
MOVL C00246 V=800.0 PL=0
MOVL C00247 V=800.0 PL=0
MOVL C00248 V=800.0 PL=0
MOVL C00249 V=800.0 PL=0
MOVL C00250 V=800.0 PL=0
MOVL C00251 V=800.0 PL=0
MOVL C00252 V=800.0 PL=0
MOVL C00253 V=800.0 PL=0
MOVL C00254 V=800.0 PL=0
MOVL C00255 V=800.0 PL=0
MOVL C00256 V=800.0 PL=0
MOVL C00257 V=800.0 PL=0
MOVL C00258 V=800.0 PL=0
MOVL C00259 V=800.0 PL=0
MOVL C00260 V=800.0 PL=0
MOVL C00261 V=800.0 PL=0
MOVL C00262 V=800.0 PL=0
MOVL C00263 V=800.0 PL=0
MOVL C00264 V=800.0 PL=0
MOVL C00265 V=800.0 PL=0
MOVL C00266 V=800.0 PL=0
MOVL C00267 V=800.0 PL=0
MOVL C00268 V=800.0 PL=0
MOVL C00269 V=800.0 PL=0
MOVL C00270 V=800.0 PL=0
MOVL C00271 V=800.0 PL=0
MOVL C00272 V=800.0 PL=0
MOVL C00273 V=800.0 PL=0
MOVL C00274 V=800.0 PL=0
MOVL C00275 V=800.0 PL=0
MOVL C00276 V=800.0 PL=0
MOVL C00277 V=800.0 PL=0
MOVL C00278 V=800.0 PL=0
MOVL C00279 V=800.0 PL=0
MOVL C00280 V=800.0 PL=0
MOVL C00281 V=800.0 PL=0
MOVL C00282 V=800.0 PL=0
MOVL C00283 V=800.0 PL=0
MOVL C00284 V=800.0 PL=0
MOVL C00285 V=800.0 PL=0
MOVL C00286 V=800.0 PL=0
MOVL C00287 V=800.0 PL=0
MOVL C00288 V=800.0 PL=0
MOVL C00289 V=800.0 PL=0
MOVL C00290 V=800.0 PL=0
MOVL C00291 V=800.0 PL=0
MOVL C00292 V=800.0 PL=0
MOVL C00293 V=800.0 PL=0
MOVL C00294 V=800.0 PL=0
MOVL C00295 V=800.0 PL=0
MOVL C00296 V=800.0 PL=0
MOVL C00297 V=800.0 PL=0
MOVL C00298 V=800.0 PL=0
MOVL C00299 V=800.0 PL=0
MOVL C00300 V=800.0 PL=0
MOVL C00301 V=800.0 PL=0
MOVL C00302 V=800.0 PL=0
MOVL C00303 V=800.0 PL=0
MOVL C00304 V=800.0 PL=0
MOVL C00305 V=800.0 PL=0
MOVL C00306 V=800.0 PL=0
MOVL C00307 V=800.0 PL=0
MOVL C00308 V=800.0 PL=0
MOVL C00309 V=800.0 PL=0
MOVL C00310 V=800.0 PL=0
MOVL C00311 V=800.0 PL=0
MOVL C00312 V=800.0 PL=0
MOVL C00313 V=800.0 PL=0
MOVL C00314 V=800.0 PL=0
MOVL C00315 V=800.0 PL=0
MOVL C00316 V=800.0 PL=0
MOVL C00317 V=800.0 PL=0
MOVL C00318 V=800.0 PL=0
MOVL C00319 V=800.0 PL=0
MOVL C00320 V=800.0 PL=0
MOVL C00321 V=800.0 PL=0
MOVL C00322 V=800.0 PL=0
MOVL C00323 V=800.0 PL=0
MOVL C00324 V=800.0 PL=0
MOVL C00325 V=800.0 PL=0
MOVL C00326 V=800.0 PL=0
MOVL C00327 V=800.0 PL=0
MOVL C00328 V=800.0 PL=0
MOVL C00329 V=800.0 PL=0
MOVL C00330 V=800.0 PL=0
MOVL C00331 V=800.0 PL=0
MOVL C00332 V=800.0 PL=0
MOVL C00333 V=800.0 PL=0
MOVL C00334 V=800.0 PL=0
MOVL C00335 V=800.0 PL=0
MOVL C00336 V=800.0 PL=0
MOVL C00337 V=800.0 PL=0
MOVL C00338 V=800.0 PL=0
MOVL C00339 V=800.0 PL=0
MOVL C00340 V=800.0 PL=0
MOVL C00341 V=800.0 PL=0
MOVL C00342 V=800.0 PL=0
MOVL C00343 V=800.0 PL=0
MOVL C00344 V=800.0 PL=0
MOVL C00345 V=800.0 PL=0
MOVL C00346 V=800.0 PL=0
MOVL C00347 V=800.0 PL=0
MOVL C00348 V=800.0 PL=0
MOVL C00349 V=800.0 PL=0
MOVL C00350 V=800.0 PL=0
MOVL C00351 V=800.0 PL=0
MOVL C00352 V=800.0 PL=0
MOVL C00353 V=800.0 PL=0
MOVL C00354 V=800.0 PL=0
MOVL C00355 V=800.0 PL=0
MOVL C00356 V=800.0 PL=0
MOVL C00357 V=800.0 PL=0
MOVL C00358 V=800.0 PL=0
MOVL C00359 V=800.0 PL=0
MOVL C00360 V=800.0 PL=0
MOVL C00361 V=800.0 PL=0
MOVL C00362 V=800.0 PL=0
MOVL C00363 V=800.0 PL=0
MOVL C00364 V=800.0 PL=0
MOVL C00365 V=800.0 PL=0
MOVL C00366 V=800.0 PL=0
MOVL C00367 V=800.0 PL=0
MOVL C00368 V=800.0 PL=0
MOVL C00369 V=800.0 PL=0
MOVL C00370 V=800.0 PL=0
MOVL C00371 V=800.0 PL=0
MOVL C00372 V=800.0 PL=0
MOVL C00373 V=800.0 PL=0
MOVL C00374 V=800.0 PL=0
MOVL C00375 V=800.0 PL=0
MOVL C00376 V=800.0 PL=0
MOVL C00377 V=800.0 PL=0
MOVL C00378 V=800.0 PL=0
MOVL C00379 V=800.0 PL=0
MOVL C00380 V=800.0 PL=0
MOVL C00381 V=800.0 PL=0
MOVL C00382 V=800.0 PL=0
MOVL C00383 V=800.0 PL=0
MOVL C00384 V=800.0 PL=0
MOVL C00385 V=800.0 PL=0
MOVL C00386 V=800.0 PL=0
MOVL C00387 V=800.0 PL=0
MOVL C00388 V=800.0 PL=0
MOVL C00389 V=800.0 PL=0
MOVL C00390 V=800.0 PL=0
MOVL C00391 V=800.0 PL=0
MOVL C00392 V=800.0 PL=0
MOVL C00393 V=800.0 PL=0
MOVL C00394 V=800.0 PL=0
MOVL C00395 V=800.0 PL=0
MOVL C00396 V=800.0 PL=0
MOVL C00397 V=800.0 PL=0
MOVL C00398 V=800.0 PL=0
MOVL C00399 V=800.0 PL=0
MOVL C00400 V=800.0 PL=0
MOVL C00401 V=800.0 PL=0
MOVL C00402 V=800.0 PL=0
MOVL C00403 V=800.0 PL=0
MOVL C00404 V=800.0 PL=0
MOVL C00405 V=800.0 PL=0
MOVL C00406 V=800.0 PL=0
MOVL C00407 V=800.0 PL=0
MOVL C00408 V=800.0 PL=0
MOVL C00409 V=800.0 PL=0
MOVL C00410 V=800.0 PL=0
MOVL C00411 V=800.0 PL=0
MOVL C00412 V=800.0 PL=0
MOVL C00413 V=800.0 PL=0
MOVL C00414 V=800.0 PL=0
MOVL C00415 V=800.0 PL=0
MOVL C00416 V=800.0 PL=0
MOVL C00417 V=800.0 PL=0
MOVL C00418 V=800.0 PL=0
MOVL C00419 V=800.0 PL=0
MOVL C00420 V=800.0 PL=0
MOVL C00421 V=800.0 PL=0
MOVL C00422 V=800.0 PL=0
MOVL C00423 V=800.0 PL=0
MOVL C00424 V=800.0 PL=0
MOVL C00425 V=800.0 PL=0
MOVL C00426 V=800.0 PL=0
MOVL C00427 V=800.0 PL=0
MOVL C00428 V=800.0 PL=0
MOVL C00429 V=800.0 PL=0
MOVL C00430 V=800.0 PL=0
MOVL C00431 V=800.0 PL=0
MOVL C00432 V=800.0 PL=0
MOVL C00433 V=800.0 PL=0
MOVL C00434 V=800.0 PL=0
MOVL C00435 V=800.0 PL=0
MOVL C00436 V=800.0 PL=0
MOVL C00437 V=800.0 PL=0
MOVL C00438 V=800.0 PL=0
MOVL C00439 V=800.0 PL=0
MOVL C00440 V=800.0 PL=0
MOVL C00441 V=800.0 PL=0
MOVL C00442 V=800.0 PL=0
MOVL C00443 V=800.0 PL=0
MOVL C00444 V=800.0 PL=0
MOVL C00445 V=800.0 PL=0
MOVL C00446 V=800.0 PL=0
MOVL C00447 V=800.0 PL=0
MOVL C00448 V=800.0 PL=0
MOVL C00449 V=800.0 PL=0
MOVL C00450 V=800.0 PL=0
MOVL C00451 V=800.0 PL=0
MOVL C00452 V=800.0 PL=0
MOVL C00453 V=800.0 PL=0
MOVL C00454 V=800.0 PL=0
MOVL C00455 V=800.0 PL=0
MOVL C00456 V=800.0 PL=0
MOVL C00457 V=800.0 PL=0
MOVL C00458 V=800.0 PL=0
MOVL C00459 V=800.0 PL=0
MOVL C00460 V=800.0 PL=0
MOVL C00461 V=800.0 PL=0
MOVL C00462 V=800.0 PL=0
MOVL C00463 V=800.0 PL=0
MOVL C00464 V=800.0 PL=0
MOVL C00465 V=800.0 PL=0
MOVL C00466 V=800.0 PL=0
MOVL C00467 V=800.0 PL=0
MOVL C00468 V=800.0 PL=0
MOVL C00469 V=800.0 PL=0
MOVL C00470 V=800.0 PL=0
MOVL C00471 V=800.0 PL=0
MOVL C00472 V=800.0 PL=0
MOVL C00473 V=800.0 PL=0
MOVL C00474 V=800.0 PL=0
MOVL C00475 V=800.0 PL=0
MOVL C00476 V=800.0 PL=0
MOVL C00477 V=800.0 PL=0
MOVL C00478 V=800.0 PL=0
MOVL C00479 V=800.0 PL=0
MOVL C00480 V=800.0 PL=0
MOVL C00481 V=800.0 PL=0
MOVL C00482 V=800.0 PL=0
MOVL C00483 V=800.0 PL=0
MOVL C00484 V=800.0 PL=0
MOVL C00485 V=800.0 PL=0
MOVL C00486 V=800.0 PL=0
MOVL C00487 V=800.0 PL=0
MOVL C00488 V=800.0 PL=0
MOVL C00489 V=800.0 PL=0
MOVL C00490 V=800.0 PL=0
MOVL C00491 V=800.0 PL=0
MOVL C00492 V=800.0 PL=0
MOVL C00493 V=800.0 PL=0
MOVL C00494 V=800.0 PL=0
MOVL C00495 V=800.0 PL=0
MOVL C00496 V=800.0 PL=0
MOVL C00497 V=800.0 PL=0
MOVL C00498 V=800.0 PL=0
MOVL C00499 V=800.0 PL=0
MOVL C00500 V=800.0 PL=0
MOVL C00501 V=800.0 PL=0
MOVL C00502 V=800.0 PL=0
MOVL C00503 V=800.0 PL=0
MOVL C00504 V=800.0 PL=0
MOVL C00505 V=800.0 PL=0
MOVL C00506 V=800.0 PL=0
MOVL C00507 V=800.0 PL=0
MOVL C00508 V=800.0 PL=0
MOVL C00509 V=800.0 PL=0
MOVL C00510 V=800.0 PL=0
MOVL C00511 V=800.0 PL=0
MOVL C00512 V=800.0 PL=0
MOVL C00513 V=800.0 PL=0
MOVL C00514 V=800.0 PL=0
MOVL C00515 V=800.0 PL=0
MOVL C00516 V=800.0 PL=0
MOVL C00517 V=800.0 PL=0
MOVL C00518 V=800.0 PL=0
MOVL C00519 V=800.0 PL=0
MOVL C00520 V=800.0 PL=0
MOVL C00521 V=800.0 PL=0
MOVL C00522 V=800.0 PL=0
MOVL C00523 V=800.0 PL=0
MOVL C00524 V=800.0 PL=0
MOVL C00525 V=800.0 PL=0
MOVL C00526 V=800.0 PL=0
MOVL C00527 V=800.0 PL=0
MOVL C00528 V=800.0 PL=0
MOVL C00529 V=800.0 PL=0
MOVL C00530 V=800.0 PL=0
MOVL C00531 V=800.0 PL=0
MOVL C00532 V=800.0 PL=0
MOVL C00533 V=800.0 PL=0
MOVL C00534 V=800.0 PL=0
MOVL C00535 V=800.0 PL=0
MOVL C00536 V=800.0 PL=0
MOVL C00537 V=800.0 PL=0
MOVL C00538 V=800.0 PL=0
MOVL C00539 V=800.0 PL=0
MOVL C00540 V=800.0 PL=0
MOVL C00541 V=800.0 PL=0
MOVL C00542 V=800.0 PL=0
MOVL C00543 V=800.0 PL=0
MOVL C00544 V=800.0 PL=0
MOVL C00545 V=800.0 PL=0
MOVL C00546 V=800.0 PL=0
MOVL C00547 V=800.0 PL=0
MOVL C00548 V=800.0 PL=0
MOVL C00549 V=800.0 PL=0
MOVL C00550 V=800.0 PL=0
MOVL C00551 V=800.0 PL=0
MOVL C00552 V=800.0 PL=0
MOVL C00553 V=800.0 PL=0
MOVL C00554 V=800.0 PL=0
MOVL C00555 V=800.0 PL=0
MOVL C00556 V=800.0 PL=0
MOVL C00557 V=800.0 PL=0
MOVL C00558 V=800.0 PL=0
MOVL C00559 V=800.0 PL=0
MOVL C00560 V=800.0 PL=0
MOVL C00561 V=800.0 PL=0
MOVL C00562 V=800.0 PL=0
MOVL C00563 V=800.0 PL=0
MOVL C00564 V=800.0 PL=0
MOVL C00565 V=800.0 PL=0
MOVL C00566 V=800.0 PL=0
MOVL C00567 V=800.0 PL=0
MOVL C00568 V=800.0 PL=0
MOVL C00569 V=800.0 PL=0
MOVL C00570 V=800.0 PL=0
MOVL C00571 V=800.0 PL=0
MOVL C00572 V=800.0 PL=0
MOVL C00573 V=800.0 PL=0
MOVL C00574 V=800.0 PL=0
MOVL C00575 V=800.0 PL=0
MOVL C00576 V=800.0 PL=0
MOVL C00577 V=800.0 PL=0
MOVL C00578 V=800.0 PL=0
MOVL C00579 V=800.0 PL=0
MOVL C00580 V=800.0 PL=0
MOVL C00581 V=800.0 PL=0
MOVL C00582 V=800.0 PL=0
MOVL C00583 V=800.0 PL=0
MOVL C00584 V=800.0 PL=0
MOVL C00585 V=800.0 PL=0
MOVL C00586 V=800.0 PL=0
MOVL C00587 V=800.0 PL=0
MOVL C00588 V=800.0 PL=0
MOVL C00589 V=800.0 PL=0
MOVL C00590 V=800.0 PL=0
MOVL C00591 V=800.0 PL=0
MOVL C00592 V=800.0 PL=0
MOVL C00593 V=800.0 PL=0
MOVL C00594 V=800.0 PL=0
MOVL C00595 V=800.0 PL=0
MOVL C00596 V=800.0 PL=0
MOVL C00597 V=800.0 PL=0
MOVL C00598 V=800.0 PL=0
MOVL C00599 V=800.0 PL=0
MOVL C00600 V=800.0 PL=0
MOVL C00601 V=800.0 PL=0
MOVL C00602 V=800.0 PL=0
MOVL C00603 V=800.0 PL=0
MOVL C00604 V=800.0 PL=0
MOVL C00605 V=800.0 PL=0
MOVL C00606 V=800.0 PL=0
MOVL C00607 V=800.0 PL=0
MOVL C00608 V=800.0 PL=0
MOVL C00609 V=800.0 PL=0
MOVL C00610 V=800.0 PL=0
MOVL C00611 V=800.0 PL=0
MOVL C00612 V=800.0 PL=0
MOVL C00613 V=800.0 PL=0
MOVL C00614 V=800.0 PL=0
MOVL C00615 V=800.0 PL=0
MOVL C00616 V=800.0 PL=0
MOVL C00617 V=800.0 PL=0
MOVL C00618 V=800.0 PL=0
MOVL C00619 V=800.0 PL=0
MOVL C00620 V=800.0 PL=0
MOVL C00621 V=800.0 PL=0
MOVL C00622 V=800.0 PL=0
MOVL C00623 V=800.0 PL=0
MOVL C00624 V=800.0 PL=0
MOVL C00625 V=800.0 PL=0
MOVL C00626 V=800.0 PL=0
MOVL C00627 V=800.0 PL=0
MOVL C00628 V=800.0 PL=0
MOVL C00629 V=800.0 PL=0
MOVL C00630 V=800.0 PL=0
MOVL C00631 V=800.0 PL=0
MOVL C00632 V=800.0 PL=0
MOVL C00633 V=800.0 PL=0
MOVL C00634 V=800.0 PL=0
MOVL C00635 V=800.0 PL=0
MOVL C00636 V=800.0 PL=0
MOVL C00637 V=800.0 PL=0
MOVL C00638 V=800.0 PL=0
MOVL C00639 V=800.0 PL=0
MOVL C00640 V=800.0 PL=0
MOVL C00641 V=800.0 PL=0
MOVL C00642 V=800.0 PL=0
MOVL C00643 V=800.0 PL=0
MOVL C00644 V=800.0 PL=0
MOVL C00645 V=800.0 PL=0
MOVL C00646 V=800.0 PL=0
MOVL C00647 V=800.0 PL=0
MOVL C00648 V=800.0 PL=0
MOVL C00649 V=800.0 PL=0
MOVL C00650 V=800.0 PL=0
MOVL C00651 V=800.0 PL=0
MOVL C00652 V=800.0 PL=0
MOVL C00653 V=800.0 PL=0
MOVL C00654 V=800.0 PL=0
MOVL C00655 V=800.0 PL=0
MOVL C00656 V=800.0 PL=0
MOVL C00657 V=800.0 PL=0
MOVL C00658 V=800.0 PL=0
MOVL C00659 V=800.0 PL=0
MOVL C00660 V=800.0 PL=0
MOVL C00661 V=800.0 PL=0
MOVL C00662 V=800.0 PL=0
MOVL C00663 V=800.0 PL=0
MOVL C00664 V=800.0 PL=0
MOVL C00665 V=800.0 PL=0
MOVL C00666 V=800.0 PL=0
MOVL C00667 V=800.0 PL=0
MOVL C00668 V=800.0 PL=0
MOVL C00669 V=800.0 PL=0
MOVL C00670 V=800.0 PL=0
MOVL C00671 V=800.0 PL=0
MOVL C00672 V=800.0 PL=0
MOVL C00673 V=800.0 PL=0
MOVL C00674 V=800.0 PL=0
MOVL C00675 V=800.0 PL=0
MOVL C00676 V=800.0 PL=0
MOVL C00677 V=800.0 PL=0
MOVL C00678 V=800.0 PL=0
MOVL C00679 V=800.0 PL=0
MOVL C00680 V=800.0 PL=0
MOVL C00681 V=800.0 PL=0
MOVL C00682 V=800.0 PL=0
MOVL C00683 V=800.0 PL=0
MOVL C00684 V=800.0 PL=0
MOVL C00685 V=800.0 PL=0
MOVL C00686 V=800.0 PL=0
MOVL C00687 V=800.0 PL=0
MOVL C00688 V=800.0 PL=0
MOVL C00689 V=800.0 PL=0
MOVL C00690 V=800.0 PL=0
MOVL C00691 V=800.0 PL=0
MOVL C00692 V=800.0 PL=0
MOVL C00693 V=800.0 PL=0
MOVL C00694 V=800.0 PL=0
MOVL C00695 V=800.0 PL=0
MOVL C00696 V=800.0 PL=0
MOVL C00697 V=800.0 PL=0
MOVL C00698 V=800.0 PL=0
MOVL C00699 V=800.0 PL=0
MOVL C00700 V=800.0 PL=0
MOVL C00701 V=800.0 PL=0
MOVL C00702 V=800.0 PL=0
MOVL C00703 V=800.0 PL=0
MOVL C00704 V=800.0 PL=0
MOVL C00705 V=800.0 PL=0
MOVL C00706 V=800.0 PL=0
MOVL C00707 V=800.0 PL=0
MOVL C00708 V=800.0 PL=0
MOVL C00709 V=800.0 PL=0
MOVL C00710 V=800.0 PL=0
MOVL C00711 V=800.0 PL=0
MOVL C00712 V=800.0 PL=0
MOVL C00713 V=800.0 PL=0
MOVL C00714 V=800.0 PL=0
MOVL C00715 V=800.0 PL=0
MOVL C00716 V=800.0 PL=0
MOVL C00717 V=800.0 PL=0
MOVL C00718 V=800.0 PL=0
MOVL C00719 V=800.0 PL=0
MOVL C00720 V=800.0 PL=0
MOVL C00721 V=800.0 PL=0
MOVL C00722 V=800.0 PL=0
MOVL C00723 V=800.0 PL=0
MOVL C00724 V=800.0 PL=0
MOVL C00725 V=800.0 PL=0
MOVL C00726 V=800.0 PL=0
MOVL C00727 V=800.0 PL=0
MOVL C00728 V=800.0 PL=0
MOVL C00729 V=800.0 PL=0
MOVL C00730 V=800.0 PL=0
MOVL C00731 V=800.0 PL=0
MOVL C00732 V=800.0 PL=0
MOVL C00733 V=800.0 PL=0
MOVL C00734 V=800.0 PL=0
MOVL C00735 V=800.0 PL=0
MOVL C00736 V=800.0 PL=0
MOVL C00737 V=800.0 PL=0
MOVL C00738 V=800.0 PL=0
MOVL C00739 V=800.0 PL=0
MOVL C00740 V=800.0 PL=0
MOVL C00741 V=800.0 PL=0
MOVL C00742 V=800.0 PL=0
MOVL C00743 V=800.0 PL=0
MOVL C00744 V=800.0 PL=0
MOVL C00745 V=800.0 PL=0
MOVL C00746 V=800.0 PL=0
MOVL C00747 V=800.0 PL=0
MOVL C00748 V=800.0 PL=0
MOVL C00749 V=800.0 PL=0
MOVL C00750 V=800.0 PL=0
MOVL C00751 V=800.0 PL=0
MOVL C00752 V=800.0 PL=0
MOVL C00753 V=800.0 PL=0
MOVL C00754 V=800.0 PL=0
MOVL C00755 V=800.0 PL=0
MOVL C00756 V=800.0 PL=0
MOVL C00757 V=800.0 PL=0
MOVL C00758 V=800.0 PL=0
MOVL C00759 V=800.0 PL=0
MOVL C00760 V=800.0 PL=0
MOVL C00761 V=800.0 PL=0
MOVL C00762 V=800.0 PL=0
MOVL C00763 V=800.0 PL=0
MOVL C00764 V=800.0 PL=0
MOVL C00765 V=800.0 PL=0
MOVL C00766 V=800.0 PL=0
MOVL C00767 V=800.0 PL=0
MOVL C00768 V=800.0 PL=0
MOVL C00769 V=800.0 PL=0
MOVL C00770 V=800.0 PL=0
MOVL C00771 V=800.0 PL=0
MOVL C00772 V=800.0 PL=0
MOVL C00773 V=800.0 PL=0
MOVL C00774 V=800.0 PL=0
MOVL C00775 V=800.0 PL=0
MOVL C00776 V=800.0 PL=0
MOVL C00777 V=800.0 PL=0
MOVL C00778 V=800.0 PL=0
MOVL C00779 V=800.0 PL=0
MOVL C00780 V=800.0 PL=0
MOVL C00781 V=800.0 PL=0
MOVL C00782 V=800.0 PL=0
MOVL C00783 V=800.0 PL=0
MOVL C00784 V=800.0 PL=0
MOVL C00785 V=800.0 PL=0
MOVL C00786 V=800.0 PL=0
MOVL C00787 V=800.0 PL=0
MOVL C00788 V=800.0 PL=0
MOVL C00789 V=800.0 PL=0
MOVL C00790 V=800.0 PL=0
MOVL C00791 V=800.0 PL=0
MOVL C00792 V=800.0 PL=0
MOVL C00793 V=800.0 PL=0
MOVL C00794 V=800.0 PL=0
MOVL C00795 V=800.0 PL=0
MOVL C00796 V=800.0 PL=0
MOVL C00797 V=800.0 PL=0
MOVL C00798 V=800.0 PL=0
MOVL C00799 V=800.0 PL=0
MOVL C00800 V=800.0 PL=0
MOVL C00801 V=800.0 PL=0
MOVL C00802 V=800.0 PL=0
MOVL C00803 V=800.0 PL=0
MOVL C00804 V=800.0 PL=0
MOVL C00805 V=800.0 PL=0
MOVL C00806 V=800.0 PL=0
MOVL C00807 V=800.0 PL=0
MOVL C00808 V=800.0 PL=0
MOVL C00809 V=800.0 PL=0
MOVL C00810 V=800.0 PL=0
MOVL C00811 V=800.0 PL=0
MOVL C00812 V=800.0 PL=0
MOVL C00813 V=800.0 PL=0
MOVL C00814 V=800.0 PL=0
MOVL C00815 V=800.0 PL=0
MOVL C00816 V=800.0 PL=0
MOVL C00817 V=800.0 PL=0
MOVL C00818 V=800.0 PL=0
MOVL C00819 V=800.0 PL=0
MOVL C00820 V=800.0 PL=0
MOVL C00821 V=800.0 PL=0
MOVL C00822 V=800.0 PL=0
MOVL C00823 V=800.0 PL=0
MOVL C00824 V=800.0 PL=0
MOVL C00825 V=800.0 PL=0
MOVL C00826 V=800.0 PL=0
MOVL C00827 V=800.0 PL=0
MOVL C00828 V=800.0 PL=0
MOVL C00829 V=800.0 PL=0
MOVL C00830 V=800.0 PL=0
MOVL C00831 V=800.0 PL=0
MOVL C00832 V=800.0 PL=0
MOVL C00833 V=800.0 PL=0
MOVL C00834 V=800.0 PL=0
MOVL C00835 V=800.0 PL=0
MOVL C00836 V=800.0 PL=0
MOVL C00837 V=800.0 PL=0
MOVL C00838 V=800.0 PL=0
MOVL C00839 V=800.0 PL=0
MOVL C00840 V=800.0 PL=0
MOVL C00841 V=800.0 PL=0
MOVL C00842 V=800.0 PL=0
MOVL C00843 V=800.0 PL=0
MOVL C00844 V=800.0 PL=0
MOVL C00845 V=800.0 PL=0
MOVL C00846 V=800.0 PL=0
MOVL C00847 V=800.0 PL=0
MOVL C00848 V=800.0 PL=0
MOVL C00849 V=800.0 PL=0
MOVL C00850 V=800.0 PL=0
MOVL C00851 V=800.0 PL=0
MOVL C00852 V=800.0 PL=0
MOVL C00853 V=800.0 PL=0
MOVL C00854 V=800.0 PL=0
MOVL C00855 V=800.0 PL=0
MOVL C00856 V=800.0 PL=0
MOVL C00857 V=800.0 PL=0
MOVL C00858 V=800.0 PL=0
MOVL C00859 V=800.0 PL=0
MOVL C00860 V=800.0 PL=0
MOVL C00861 V=800.0 PL=0
MOVL C00862 V=800.0 PL=0
MOVL C00863 V=800.0 PL=0
MOVL C00864 V=800.0 PL=0
MOVL C00865 V=800.0 PL=0
MOVL C00866 V=800.0 PL=0
MOVL C00867 V=800.0 PL=0
MOVL C00868 V=800.0 PL=0
MOVL C00869 V=800.0 PL=0
MOVL C00870 V=800.0 PL=0
MOVL C00871 V=800.0 PL=0
MOVL C00872 V=800.0 PL=0
MOVL C00873 V=800.0 PL=0
MOVL C00874 V=800.0 PL=0
MOVL C00875 V=800.0 PL=0
MOVL C00876 V=800.0 PL=0
MOVL C00877 V=800.0 PL=0
MOVL C00878 V=800.0 PL=0
MOVL C00879 V=800.0 PL=0
MOVL C00880 V=800.0 PL=0
MOVL C00881 V=800.0 PL=0
MOVL C00882 V=800.0 PL=0
MOVL C00883 V=800.0 PL=0
MOVL C00884 V=800.0 PL=0
MOVL C00885 V=800.0 PL=0
MOVL C00886 V=800.0 PL=0
MOVL C00887 V=800.0 PL=0
MOVL C00888 V=800.0 PL=0
MOVL C00889 V=800.0 PL=0
MOVL C00890 V=800.0 PL=0
MOVL C00891 V=800.0 PL=0
MOVL C00892 V=800.0 PL=0
MOVL C00893 V=800.0 PL=0
MOVL C00894 V=800.0 PL=0
MOVL C00895 V=800.0 PL=0
MOVL C00896 V=800.0 PL=0
MOVL C00897 V=800.0 PL=0
MOVL C00898 V=800.0 PL=0
MOVL C00899 V=800.0 PL=0
MOVL C00900 V=800.0 PL=0
MOVL C00901 V=800.0 PL=0
MOVL C00902 V=800.0 PL=0
MOVL C00903 V=800.0 PL=0
MOVL C00904 V=800.0 PL=0
MOVL C00905 V=800.0 PL=0
MOVL C00906 V=800.0 PL=0
MOVL C00907 V=800.0 PL=0
MOVL C00908 V=800.0 PL=0
MOVL C00909 V=800.0 PL=0
MOVL C00910 V=800.0 PL=0
MOVL C00911 V=800.0 PL=0
MOVL C00912 V=800.0 PL=0
MOVL C00913 V=800.0 PL=0
MOVL C00914 V=800.0 PL=0
MOVL C00915 V=800.0 PL=0
MOVL C00916 V=800.0 PL=0
MOVL C00917 V=800.0 PL=0
MOVL C00918 V=800.0 PL=0
MOVL C00919 V=800.0 PL=0
MOVL C00920 V=800.0 PL=0
MOVL C00921 V=800.0 PL=0
MOVL C00922 V=800.0 PL=0
MOVL C00923 V=800.0 PL=0
MOVL C00924 V=800.0 PL=0
MOVL C00925 V=800.0 PL=0
MOVL C00926 V=800.0 PL=0
MOVL C00927 V=800.0 PL=0
MOVL C00928 V=800.0 PL=0
MOVL C00929 V=800.0 PL=0
MOVL C00930 V=800.0 PL=0
MOVL C00931 V=800.0 PL=0
MOVL C00932 V=800.0 PL=0
MOVL C00933 V=800.0 PL=0
MOVL C00934 V=800.0 PL=0
MOVL C00935 V=800.0 PL=0
MOVL C00936 V=800.0 PL=0
MOVL C00937 V=800.0 PL=0
MOVL C00938 V=800.0 PL=0
MOVL C00939 V=800.0 PL=0
MOVL C00940 V=800.0 PL=0
MOVL C00941 V=800.0 PL=0
MOVL C00942 V=800.0 PL=0
MOVL C00943 V=800.0 PL=0
MOVL C00944 V=800.0 PL=0
MOVL C00945 V=800.0 PL=0
MOVL C00946 V=800.0 PL=0
MOVL C00947 V=800.0 PL=0
MOVL C00948 V=800.0 PL=0
MOVL C00949 V=800.0 PL=0
MOVL C00950 V=800.0 PL=0
MOVL C00951 V=800.0 PL=0
MOVL C00952 V=800.0 PL=0
MOVL C00953 V=800.0 PL=0
MOVL C00954 V=800.0 PL=0
MOVL C00955 V=800.0 PL=0
MOVL C00956 V=800.0 PL=0
MOVL C00957 V=800.0 PL=0
MOVL C00958 V=800.0 PL=0
MOVL C00959 V=800.0 PL=0
MOVL C00960 V=800.0 PL=0
MOVL C00961 V=800.0 PL=0
MOVL C00962 V=800.0 PL=0
MOVL C00963 V=800.0 PL=0
MOVL C00964 V=800.0 PL=0
MOVL C00965 V=800.0 PL=0
MOVL C00966 V=800.0 PL=0
MOVL C00967 V=800.0 PL=0
MOVL C00968 V=800.0 PL=0
MOVL C00969 V=800.0 PL=0
MOVL C00970 V=800.0 PL=0
MOVL C00971 V=800.0 PL=0
MOVL C00972 V=800.0 PL=0
MOVL C00973 V=800.0 PL=0
MOVL C00974 V=800.0 PL=0
MOVL C00975 V=800.0 PL=0
MOVL C00976 V=800.0 PL=0
MOVL C00977 V=800.0 PL=0
MOVL C00978 V=800.0 PL=0
MOVL C00979 V=800.0 PL=0
MOVL C00980 V=800.0 PL=0
MOVL C00981 V=800.0 PL=0
MOVL C00982 V=800.0 PL=0
MOVL C00983 V=800.0 PL=0
MOVL C00984 V=800.0 PL=0
MOVL C00985 V=800.0 PL=0
MOVL C00986 V=800.0 PL=0
MOVL C00987 V=800.0 PL=0
MOVL C00988 V=800.0 PL=0
MOVL C00989 V=800.0 PL=0
MOVL C00990 V=800.0 PL=0
MOVL C00991 V=800.0 PL=0
MOVL C00992 V=800.0 PL=0
MOVL C00993 V=800.0 PL=0
MOVL C00994 V=800.0 PL=0
MOVL C00995 V=800.0 PL=0
MOVL C00996 V=800.0 PL=0
MOVL C00997 V=800.0 PL=0
MOVL C00998 V=800.0 PL=0
MOVL C00999 V=800.0 PL=0
MOVL C01000 V=800.0 PL=0
MOVL C01001 V=800.0 PL=0
MOVL C01002 V=800.0 PL=0
MOVL C01003 V=800.0 PL=0
MOVL C01004 V=800.0 PL=0
MOVL C01005 V=800.0 PL=0
MOVL C01006 V=800.0 PL=0
MOVL C01007 V=800.0 PL=0
MOVL C01008 V=800.0 PL=0
MOVL C01009 V=800.0 PL=0
MOVL C01010 V=800.0 PL=0
MOVL C01011 V=800.0 PL=0
MOVL C01012 V=800.0 PL=0
MOVL C01013 V=800.0 PL=0
MOVL C01014 V=800.0 PL=0
MOVL C01015 V=800.0 PL=0
MOVL C01016 V=800.0 PL=0
MOVL C01017 V=800.0 PL=0
MOVL C01018 V=800.0 PL=0
MOVL C01019 V=800.0 PL=0
MOVL C01020 V=800.0 PL=0
MOVL C01021 V=800.0 PL=0
MOVL C01022 V=800.0 PL=0
MOVL C01023 V=800.0 PL=0
MOVL C01024 V=800.0 PL=0
MOVL C01025 V=800.0 PL=0
MOVL C01026 V=800.0 PL=0
MOVL C01027 V=800.0 PL=0
MOVL C01028 V=800.0 PL=0
MOVL C01029 V=800.0 PL=0
MOVL C01030 V=800.0 PL=0
MOVL C01031 V=800.0 PL=0
MOVL C01032 V=800.0 PL=0
MOVL C01033 V=800.0 PL=0
MOVL C01034 V=800.0 PL=0
MOVL C01035 V=800.0 PL=0
MOVL C01036 V=800.0 PL=0
MOVL C01037 V=800.0 PL=0
MOVL C01038 V=800.0 PL=0
MOVL C01039 V=800.0 PL=0
MOVL C01040 V=800.0 PL=0
MOVL C01041 V=800.0 PL=0
MOVL C01042 V=800.0 PL=0
MOVL C01043 V=800.0 PL=0
MOVL C01044 V=800.0 PL=0
MOVL C01045 V=800.0 PL=0
MOVL C01046 V=800.0 PL=0
MOVL C01047 V=800.0 PL=0
MOVL C01048 V=800.0 PL=0
MOVL C01049 V=800.0 PL=0
MOVL C01050 V=800.0 PL=0
MOVL C01051 V=800.0 PL=0
MOVL C01052 V=800.0 PL=0
MOVL C01053 V=800.0 PL=0
MOVL C01054 V=800.0 PL=0
MOVL C01055 V=800.0 PL=0
MOVL C01056 V=800.0 PL=0
MOVL C01057 V=800.0 PL=0
MOVL C01058 V=800.0 PL=0
MOVL C01059 V=800.0 PL=0
MOVL C01060 V=800.0 PL=0
MOVL C01061 V=800.0 PL=0
MOVL C01062 V=800.0 PL=0
MOVL C01063 V=800.0 PL=0
MOVL C01064 V=800.0 PL=0
MOVL C01065 V=800.0 PL=0
MOVL C01066 V=800.0 PL=0
MOVL C01067 V=800.0 PL=0
MOVL C01068 V=800.0 PL=0
MOVL C01069 V=800.0 PL=0
MOVL C01070 V=800.0 PL=0
MOVL C01071 V=800.0 PL=0
MOVL C01072 V=800.0 PL=0
MOVL C01073 V=800.0 PL=0
MOVL C01074 V=800.0 PL=0
MOVL C01075 V=800.0 PL=0
MOVL C01076 V=800.0 PL=0
MOVL C01077 V=800.0 PL=0
MOVL C01078 V=800.0 PL=0
MOVL C01079 V=800.0 PL=0
MOVL C01080 V=800.0 PL=0
MOVL C01081 V=800.0 PL=0
MOVL C01082 V=800.0 PL=0
MOVL C01083 V=800.0 PL=0
MOVL C01084 V=800.0 PL=0
MOVL C01085 V=800.0 PL=0
MOVL C01086 V=800.0 PL=0
MOVL C01087 V=800.0 PL=0
MOVL C01088 V=800.0 PL=0
MOVL C01089 V=800.0 PL=0
MOVL C01090 V=800.0 PL=0
MOVL C01091 V=800.0 PL=0
MOVL C01092 V=800.0 PL=0
MOVL C01093 V=800.0 PL=0
MOVL C01094 V=800.0 PL=0
MOVL C01095 V=800.0 PL=0
MOVL C01096 V=800.0 PL=0
MOVL C01097 V=800.0 PL=0
MOVL C01098 V=800.0 PL=0
MOVL C01099 V=800.0 PL=0
MOVL C01100 V=800.0 PL=0
MOVL C01101 V=800.0 PL=0
MOVL C01102 V=800.0 PL=0
MOVL C01103 V=800.0 PL=0
MOVL C01104 V=800.0 PL=0
MOVL C01105 V=800.0 PL=0
MOVL C01106 V=800.0 PL=0
MOVL C01107 V=800.0 PL=0
MOVL C01108 V=800.0 PL=0
MOVL C01109 V=800.0 PL=0
MOVL C01110 V=800.0 PL=0
MOVL C01111 V=800.0 PL=0
MOVL C01112 V=800.0 PL=0
MOVL C01113 V=800.0 PL=0
MOVL C01114 V=800.0 PL=0
MOVL C01115 V=800.0 PL=0
MOVL C01116 V=800.0 PL=0
MOVL C01117 V=800.0 PL=0
MOVL C01118 V=800.0 PL=0
MOVL C01119 V=800.0 PL=0
MOVL C01120 V=800.0 PL=0
MOVL C01121 V=800.0 PL=0
MOVL C01122 V=800.0 PL=0
MOVL C01123 V=800.0 PL=0
MOVL C01124 V=800.0 PL=0
MOVL C01125 V=800.0 PL=0
MOVL C01126 V=800.0 PL=0
MOVL C01127 V=800.0 PL=0
MOVL C01128 V=800.0 PL=0
MOVL C01129 V=800.0 PL=0
MOVL C01130 V=800.0 PL=0
MOVL C01131 V=800.0 PL=0
MOVL C01132 V=800.0 PL=0
MOVL C01133 V=800.0 PL=0
MOVL C01134 V=800.0 PL=0
MOVL C01135 V=800.0 PL=0
MOVL C01136 V=800.0 PL=0
MOVL C01137 V=800.0 PL=0
MOVL C01138 V=800.0 PL=0
MOVL C01139 V=800.0 PL=0
MOVL C01140 V=800.0 PL=0
MOVL C01141 V=800.0 PL=0
MOVL C01142 V=800.0 PL=0
MOVL C01143 V=800.0 PL=0
MOVL C01144 V=800.0 PL=0
MOVL C01145 V=800.0 PL=0
MOVL C01146 V=800.0 PL=0
MOVL C01147 V=800.0 PL=0
MOVL C01148 V=800.0 PL=0
MOVL C01149 V=800.0 PL=0
MOVL C01150 V=800.0 PL=0
MOVL C01151 V=800.0 PL=0
MOVL C01152 V=800.0 PL=0
MOVL C01153 V=800.0 PL=0
MOVL C01154 V=800.0 PL=0
MOVL C01155 V=800.0 PL=0
MOVL C01156 V=800.0 PL=0
MOVL C01157 V=800.0 PL=0
MOVL C01158 V=800.0 PL=0
MOVL C01159 V=800.0 PL=0
MOVL C01160 V=800.0 PL=0
MOVL C01161 V=800.0 PL=0
MOVL C01162 V=800.0 PL=0
MOVL C01163 V=800.0 PL=0
MOVL C01164 V=800.0 PL=0
MOVL C01165 V=800.0 PL=0
MOVL C01166 V=800.0 PL=0
MOVL C01167 V=800.0 PL=0
MOVL C01168 V=800.0 PL=0
MOVL C01169 V=800.0 PL=0
MOVL C01170 V=800.0 PL=0
MOVL C01171 V=800.0 PL=0
MOVL C01172 V=800.0 PL=0
MOVL C01173 V=800.0 PL=0
MOVL C01174 V=800.0 PL=0
MOVL C01175 V=800.0 PL=0
MOVL C01176 V=800.0 PL=0
MOVL C01177 V=800.0 PL=0
MOVL C01178 V=800.0 PL=0
MOVL C01179 V=800.0 PL=0
MOVL C01180 V=800.0 PL=0
MOVL C01181 V=800.0 PL=0
MOVL C01182 V=800.0 PL=0
MOVL C01183 V=800.0 PL=0
MOVL C01184 V=800.0 PL=0
MOVL C01185 V=800.0 PL=0
MOVL C01186 V=800.0 PL=0
MOVL C01187 V=800.0 PL=0
MOVL C01188 V=800.0 PL=0
MOVL C01189 V=800.0 PL=0
MOVL C01190 V=800.0 PL=0
MOVL C01191 V=800.0 PL=0
MOVL C01192 V=800.0 PL=0
MOVL C01193 V=800.0 PL=0
MOVL C01194 V=800.0 PL=0
MOVL C01195 V=800.0 PL=0
MOVL C01196 V=800.0 PL=0
MOVL C01197 V=800.0 PL=0
MOVL C01198 V=800.0 PL=0
MOVL C01199 V=800.0 PL=0
MOVL C01200 V=800.0 PL=0
MOVL C01201 V=800.0 PL=0
MOVL C01202 V=800.0 PL=0
MOVL C01203 V=800.0 PL=0
MOVL C01204 V=800.0 PL=0
MOVL C01205 V=800.0 PL=0
MOVL C01206 V=800.0 PL=0
MOVL C01207 V=800.0 PL=0
MOVL C01208 V=800.0 PL=0
MOVL C01209 V=800.0 PL=0
MOVL C01210 V=800.0 PL=0
MOVL C01211 V=800.0 PL=0
MOVL C01212 V=800.0 PL=0
MOVL C01213 V=800.0 PL=0
MOVL C01214 V=800.0 PL=0
MOVL C01215 V=800.0 PL=0
MOVL C01216 V=800.0 PL=0
MOVL C01217 V=800.0 PL=0
MOVL C01218 V=800.0 PL=0
MOVL C01219 V=800.0 PL=0
MOVL C01220 V=800.0 PL=0
MOVL C01221 V=800.0 PL=0
MOVL C01222 V=800.0 PL=0
MOVL C01223 V=800.0 PL=0
MOVL C01224 V=800.0 PL=0
MOVL C01225 V=800.0 PL=0
MOVL C01226 V=800.0 PL=0
MOVL C01227 V=800.0 PL=0
MOVL C01228 V=800.0 PL=0
MOVL C01229 V=800.0 PL=0
MOVL C01230 V=800.0 PL=0
MOVL C01231 V=800.0 PL=0
MOVL C01232 V=800.0 PL=0
MOVL C01233 V=800.0 PL=0
MOVL C01234 V=800.0 PL=0
MOVL C01235 V=800.0 PL=0
MOVL C01236 V=800.0 PL=0
MOVL C01237 V=800.0 PL=0
MOVL C01238 V=800.0 PL=0
MOVL C01239 V=800.0 PL=0
MOVL C01240 V=800.0 PL=0
MOVL C01241 V=800.0 PL=0
MOVL C01242 V=800.0 PL=0
MOVL C01243 V=800.0 PL=0
MOVL C01244 V=800.0 PL=0
MOVL C01245 V=800.0 PL=0
MOVL C01246 V=800.0 PL=0
MOVL C01247 V=800.0 PL=0
MOVL C01248 V=800.0 PL=0
MOVL C01249 V=800.0 PL=0
MOVL C01250 V=800.0 PL=0
MOVL C01251 V=800.0 PL=0
MOVL C01252 V=800.0 PL=0
MOVL C01253 V=800.0 PL=0
MOVL C01254 V=800.0 PL=0
MOVL C01255 V=800.0 PL=0
MOVL C01256 V=800.0 PL=0
MOVL C01257 V=800.0 PL=0
MOVL C01258 V=800.0 PL=0
MOVL C01259 V=800.0 PL=0
MOVL C01260 V=800.0 PL=0
MOVL C01261 V=800.0 PL=0
MOVL C01262 V=800.0 PL=0
MOVL C01263 V=800.0 PL=0
MOVL C01264 V=800.0 PL=0
MOVL C01265 V=800.0 PL=0
MOVL C01266 V=800.0 PL=0
MOVL C01267 V=800.0 PL=0
MOVL C01268 V=800.0 PL=0
MOVL C01269 V=800.0 PL=0
MOVL C01270 V=800.0 PL=0
MOVL C01271 V=800.0 PL=0
MOVL C01272 V=800.0 PL=0
MOVL C01273 V=800.0 PL=0
MOVL C01274 V=800.0 PL=0
MOVL C01275 V=800.0 PL=0
MOVL C01276 V=800.0 PL=0
MOVL C01277 V=800.0 PL=0
MOVL C01278 V=800.0 PL=0
MOVL C01279 V=800.0 PL=0
MOVL C01280 V=800.0 PL=0
MOVL C01281 V=800.0 PL=0
MOVL C01282 V=800.0 PL=0
MOVL C01283 V=800.0 PL=0
MOVL C01284 V=800.0 PL=0
MOVL C01285 V=800.0 PL=0
MOVL C01286 V=800.0 PL=0
MOVL C01287 V=800.0 PL=0
MOVL C01288 V=800.0 PL=0
MOVL C01289 V=800.0 PL=0
MOVL C01290 V=800.0 PL=0
MOVL C01291 V=800.0 PL=0
MOVL C01292 V=800.0 PL=0
MOVL C01293 V=800.0 PL=0
MOVL C01294 V=800.0 PL=0
MOVL C01295 V=800.0 PL=0
MOVL C01296 V=800.0 PL=0
MOVL C01297 V=800.0 PL=0
MOVL C01298 V=800.0 PL=0
MOVL C01299 V=800.0 PL=0
MOVL C01300 V=800.0 PL=0
MOVL C01301 V=800.0 PL=0
MOVL C01302 V=800.0 PL=0
MOVL C01303 V=800.0 PL=0
MOVL C01304 V=800.0 PL=0
MOVL C01305 V=800.0 PL=0
MOVL C01306 V=800.0 PL=0
MOVL C01307 V=800.0 PL=0
MOVL C01308 V=800.0 PL=0
MOVL C01309 V=800.0 PL=0
MOVL C01310 V=800.0 PL=0
MOVL C01311 V=800.0 PL=0
MOVL C01312 V=800.0 PL=0
MOVL C01313 V=800.0 PL=0
MOVL C01314 V=800.0 PL=0
MOVL C01315 V=800.0 PL=0
MOVL C01316 V=800.0 PL=0
MOVL C01317 V=800.0 PL=0
MOVL C01318 V=800.0 PL=0
MOVL C01319 V=800.0 PL=0
MOVL C01320 V=800.0 PL=0
MOVL C01321 V=800.0 PL=0
MOVL C01322 V=800.0 PL=0
MOVL C01323 V=800.0 PL=0
MOVL C01324 V=800.0 PL=0
MOVL C01325 V=800.0 PL=0
MOVL C01326 V=800.0 PL=0
MOVL C01327 V=800.0 PL=0
MOVL C01328 V=800.0 PL=0
MOVL C01329 V=800.0 PL=0
MOVL C01330 V=800.0 PL=0
MOVL C01331 V=800.0 PL=0
MOVL C01332 V=800.0 PL=0
MOVL C01333 V=800.0 PL=0
MOVL C01334 V=800.0 PL=0
MOVL C01335 V=800.0 PL=0
MOVL C01336 V=800.0 PL=0
MOVL C01337 V=800.0 PL=0
MOVL C01338 V=800.0 PL=0
MOVL C01339 V=800.0 PL=0
MOVL C01340 V=800.0 PL=0
MOVL C01341 V=800.0 PL=0
MOVL C01342 V=800.0 PL=0
MOVL C01343 V=800.0 PL=0
MOVL C01344 V=800.0 PL=0
MOVL C01345 V=800.0 PL=0
MOVL C01346 V=800.0 PL=0
MOVL C01347 V=800.0 PL=0
MOVL C01348 V=800.0 PL=0
MOVL C01349 V=800.0 PL=0
MOVL C01350 V=800.0 PL=0
MOVL C01351 V=800.0 PL=0
MOVL C01352 V=800.0 PL=0
MOVL C01353 V=800.0 PL=0
MOVL C01354 V=800.0 PL=0
MOVL C01355 V=800.0 PL=0
MOVL C01356 V=800.0 PL=0
MOVL C01357 V=800.0 PL=0
MOVL C01358 V=800.0 PL=0
MOVL C01359 V=800.0 PL=0
MOVL C01360 V=800.0 PL=0
MOVL C01361 V=800.0 PL=0
MOVL C01362 V=800.0 PL=0
MOVL C01363 V=800.0 PL=0
MOVL C01364 V=800.0 PL=0
MOVL C01365 V=800.0 PL=0
MOVL C01366 V=800.0 PL=0
MOVL C01367 V=800.0 PL=0
MOVL C01368 V=800.0 PL=0
MOVL C01369 V=800.0 PL=0
MOVL C01370 V=800.0 PL=0
MOVL C01371 V=800.0 PL=0
MOVL C01372 V=800.0 PL=0
MOVL C01373 V=800.0 PL=0
MOVL C01374 V=800.0 PL=0
MOVL C01375 V=800.0 PL=0
MOVL C01376 V=800.0 PL=0
MOVL C01377 V=800.0 PL=0
MOVL C01378 V=800.0 PL=0
MOVL C01379 V=800.0 PL=0
MOVL C01380 V=800.0 PL=0
MOVL C01381 V=800.0 PL=0
MOVL C01382 V=800.0 PL=0
MOVL C01383 V=800.0 PL=0
MOVL C01384 V=800.0 PL=0
MOVL C01385 V=800.0 PL=0
MOVL C01386 V=800.0 PL=0
MOVL C01387 V=800.0 PL=0
MOVL C01388 V=800.0 PL=0
MOVL C01389 V=800.0 PL=0
MOVL C01390 V=800.0 PL=0
MOVL C01391 V=800.0 PL=0
MOVL C01392 V=800.0 PL=0
MOVL C01393 V=800.0 PL=0
MOVL C01394 V=800.0 PL=0
MOVL C01395 V=800.0 PL=0
MOVL C01396 V=800.0 PL=0
MOVL C01397 V=800.0 PL=0
MOVL C01398 V=800.0 PL=0
MOVL C01399 V=800.0 PL=0
MOVL C01400 V=800.0 PL=0
MOVL C01401 V=800.0 PL=0
MOVL C01402 V=800.0 PL=0
MOVL C01403 V=800.0 PL=0
MOVL C01404 V=800.0 PL=0
MOVL C01405 V=800.0 PL=0
MOVL C01406 V=800.0 PL=0
MOVL C01407 V=800.0 PL=0
MOVL C01408 V=800.0 PL=0
MOVL C01409 V=800.0 PL=0
MOVL C01410 V=800.0 PL=0
MOVL C01411 V=800.0 PL=0
MOVL C01412 V=800.0 PL=0
MOVL C01413 V=800.0 PL=0
MOVL C01414 V=800.0 PL=0
MOVL C01415 V=800.0 PL=0
MOVL C01416 V=800.0 PL=0
MOVL C01417 V=800.0 PL=0
MOVL C01418 V=800.0 PL=0
MOVL C01419 V=800.0 PL=0
MOVL C01420 V=800.0 PL=0
MOVL C01421 V=800.0 PL=0
MOVL C01422 V=800.0 PL=0
MOVL C01423 V=800.0 PL=0
MOVL C01424 V=800.0 PL=0
MOVL C01425 V=800.0 PL=0
MOVL C01426 V=800.0 PL=0
MOVL C01427 V=800.0 PL=0
MOVL C01428 V=800.0 PL=0
MOVL C01429 V=800.0 PL=0
MOVL C01430 V=800.0 PL=0
MOVL C01431 V=800.0 PL=0
MOVL C01432 V=800.0 PL=0
MOVL C01433 V=800.0 PL=0
MOVL C01434 V=800.0 PL=0
MOVL C01435 V=800.0 PL=0
MOVL C01436 V=800.0 PL=0
MOVL C01437 V=800.0 PL=0
MOVL C01438 V=800.0 PL=0
MOVL C01439 V=800.0 PL=0
MOVL C01440 V=800.0 PL=0
MOVL C01441 V=800.0 PL=0
MOVL C01442 V=800.0 PL=0
MOVL C01443 V=800.0 PL=0
MOVL C01444 V=800.0 PL=0
MOVL C01445 V=800.0 PL=0
MOVL C01446 V=800.0 PL=0
MOVL C01447 V=800.0 PL=0
MOVL C01448 V=800.0 PL=0
MOVL C01449 V=800.0 PL=0
MOVL C01450 V=800.0 PL=0
MOVL C01451 V=800.0 PL=0
MOVL C01452 V=800.0 PL=0
MOVL C01453 V=800.0 PL=0
MOVL C01454 V=800.0 PL=0
MOVL C01455 V=800.0 PL=0
MOVL C01456 V=800.0 PL=0
MOVL C01457 V=800.0 PL=0
MOVL C01458 V=800.0 PL=0
MOVL C01459 V=800.0 PL=0
MOVL C01460 V=800.0 PL=0
MOVL C01461 V=800.0 PL=0
MOVL C01462 V=800.0 PL=0
MOVL C01463 V=800.0 PL=0
MOVL C01464 V=800.0 PL=0
MOVL C01465 V=800.0 PL=0
MOVL C01466 V=800.0 PL=0
MOVL C01467 V=800.0 PL=0
MOVL C01468 V=800.0 PL=0
MOVL C01469 V=800.0 PL=0
MOVL C01470 V=800.0 PL=0
MOVL C01471 V=800.0 PL=0
MOVL C01472 V=800.0 PL=0
MOVL C01473 V=800.0 PL=0
MOVL C01474 V=800.0 PL=0
MOVL C01475 V=800.0 PL=0
MOVL C01476 V=800.0 PL=0
MOVL C01477 V=800.0 PL=0
MOVL C01478 V=800.0 PL=0
MOVL C01479 V=800.0 PL=0
MOVL C01480 V=800.0 PL=0
MOVL C01481 V=800.0 PL=0
MOVL C01482 V=800.0 PL=0
MOVL C01483 V=800.0 PL=0
MOVL C01484 V=800.0 PL=0
MOVL C01485 V=800.0 PL=0
MOVL C01486 V=800.0 PL=0
MOVL C01487 V=800.0 PL=0
MOVL C01488 V=800.0 PL=0
MOVL C01489 V=800.0 PL=0
MOVL C01490 V=800.0 PL=0
MOVL C01491 V=800.0 PL=0
MOVL C01492 V=800.0 PL=0
MOVL C01493 V=800.0 PL=0
MOVL C01494 V=800.0 PL=0
MOVL C01495 V=800.0 PL=0
MOVL C01496 V=800.0 PL=0
MOVL C01497 V=800.0 PL=0
MOVL C01498 V=800.0 PL=0
MOVL C01499 V=800.0 PL=0
MOVL C01500 V=800.0 PL=0
MOVL C01501 V=800.0 PL=0
MOVL C01502 V=800.0 PL=0
MOVL C01503 V=800.0 PL=0
MOVL C01504 V=800.0 PL=0
MOVL C01505 V=800.0 PL=0
MOVL C01506 V=800.0 PL=0
MOVL C01507 V=800.0 PL=0
MOVL C01508 V=800.0 PL=0
MOVL C01509 V=800.0 PL=0
MOVL C01510 V=800.0 PL=0
MOVL C01511 V=800.0 PL=0
MOVL C01512 V=800.0 PL=0
MOVL C01513 V=800.0 PL=0
MOVL C01514 V=800.0 PL=0
MOVL C01515 V=800.0 PL=0
MOVL C01516 V=800.0 PL=0
MOVL C01517 V=800.0 PL=0
MOVL C01518 V=800.0 PL=0
MOVL C01519 V=800.0 PL=0
MOVL C01520 V=800.0 PL=0
MOVL C01521 V=800.0 PL=0
MOVL C01522 V=800.0 PL=0
MOVL C01523 V=800.0 PL=0
MOVL C01524 V=800.0 PL=0
MOVL C01525 V=800.0 PL=0
MOVL C01526 V=800.0 PL=0
MOVL C01527 V=800.0 PL=0
MOVL C01528 V=800.0 PL=0
MOVL C01529 V=800.0 PL=0
MOVL C01530 V=800.0 PL=0
MOVL C01531 V=800.0 PL=0
MOVL C01532 V=800.0 PL=0
MOVL C01533 V=800.0 PL=0
MOVL C01534 V=800.0 PL=0
MOVL C01535 V=800.0 PL=0
MOVL C01536 V=800.0 PL=0
MOVL C01537 V=800.0 PL=0
MOVL C01538 V=800.0 PL=0
MOVL C01539 V=800.0 PL=0
MOVL C01540 V=800.0 PL=0
MOVL C01541 V=800.0 PL=0
MOVL C01542 V=800.0 PL=0
MOVL C01543 V=800.0 PL=0
MOVL C01544 V=800.0 PL=0
MOVL C01545 V=800.0 PL=0
MOVL C01546 V=800.0 PL=0
MOVL C01547 V=800.0 PL=0
MOVL C01548 V=800.0 PL=0
MOVL C01549 V=800.0 PL=0
MOVL C01550 V=800.0 PL=0
MOVL C01551 V=800.0 PL=0
MOVL C01552 V=800.0 PL=0
MOVL C01553 V=800.0 PL=0
MOVL C01554 V=800.0 PL=0
MOVL C01555 V=800.0 PL=0
MOVL C01556 V=800.0 PL=0
MOVL C01557 V=800.0 PL=0
MOVL C01558 V=800.0 PL=0
MOVL C01559 V=800.0 PL=0
MOVL C01560 V=800.0 PL=0
MOVL C01561 V=800.0 PL=0
MOVL C01562 V=800.0 PL=0
MOVL C01563 V=800.0 PL=0
MOVL C01564 V=800.0 PL=0
MOVL C01565 V=800.0 PL=0
MOVL C01566 V=800.0 PL=0
MOVL C01567 V=800.0 PL=0
MOVL C01568 V=800.0 PL=0
MOVL C01569 V=800.0 PL=0
MOVL C01570 V=800.0 PL=0
MOVL C01571 V=800.0 PL=0
MOVL C01572 V=800.0 PL=0
MOVL C01573 V=800.0 PL=0
MOVL C01574 V=800.0 PL=0
MOVL C01575 V=800.0 PL=0
MOVL C01576 V=800.0 PL=0
MOVL C01577 V=800.0 PL=0
MOVL C01578 V=800.0 PL=0
MOVL C01579 V=800.0 PL=0
MOVL C01580 V=800.0 PL=0
MOVL C01581 V=800.0 PL=0
MOVL C01582 V=800.0 PL=0
MOVL C01583 V=800.0 PL=0
MOVL C01584 V=800.0 PL=0
MOVL C01585 V=800.0 PL=0
MOVL C01586 V=800.0 PL=0
MOVL C01587 V=800.0 PL=0
MOVL C01588 V=800.0 PL=0
MOVL C01589 V=800.0 PL=0
MOVL C01590 V=800.0 PL=0
MOVL C01591 V=800.0 PL=0
MOVL C01592 V=800.0 PL=0
MOVL C01593 V=800.0 PL=0
MOVL C01594 V=800.0 PL=0
MOVL C01595 V=800.0 PL=0
MOVL C01596 V=800.0 PL=0
MOVL C01597 V=800.0 PL=0
MOVL C01598 V=800.0 PL=0
MOVL C01599 V=800.0 PL=0
MOVL C01600 V=800.0 PL=0
MOVL C01601 V=800.0 PL=0
MOVL C01602 V=800.0 PL=0
MOVL C01603 V=800.0 PL=0
MOVL C01604 V=800.0 PL=0
MOVL C01605 V=800.0 PL=0
MOVL C01606 V=800.0 PL=0
MOVL C01607 V=800.0 PL=0
MOVL C01608 V=800.0 PL=0
MOVL C01609 V=800.0 PL=0
MOVL C01610 V=800.0 PL=0
MOVL C01611 V=800.0 PL=0
MOVL C01612 V=800.0 PL=0
MOVL C01613 V=800.0 PL=0
MOVL C01614 V=800.0 PL=0
MOVL C01615 V=800.0 PL=0
MOVL C01616 V=800.0 PL=0
MOVL C01617 V=800.0 PL=0
MOVL C01618 V=800.0 PL=0
MOVL C01619 V=800.0 PL=0
MOVL C01620 V=800.0 PL=0
MOVL C01621 V=800.0 PL=0
MOVL C01622 V=800.0 PL=0
MOVL C01623 V=800.0 PL=0
MOVL C01624 V=800.0 PL=0
MOVL C01625 V=800.0 PL=0
MOVL C01626 V=800.0 PL=0
MOVL C01627 V=800.0 PL=0
MOVL C01628 V=800.0 PL=0
MOVL C01629 V=800.0 PL=0
MOVL C01630 V=800.0 PL=0
MOVL C01631 V=800.0 PL=0
MOVL C01632 V=800.0 PL=0
MOVL C01633 V=800.0 PL=0
MOVL C01634 V=800.0 PL=0
MOVL C01635 V=800.0 PL=0
MOVL C01636 V=800.0 PL=0
MOVL C01637 V=800.0 PL=0
MOVL C01638 V=800.0 PL=0
MOVL C01639 V=800.0 PL=0
MOVL C01640 V=800.0 PL=0
MOVL C01641 V=800.0 PL=0
MOVL C01642 V=800.0 PL=0
MOVL C01643 V=800.0 PL=0
MOVL C01644 V=800.0 PL=0
MOVL C01645 V=800.0 PL=0
MOVL C01646 V=800.0 PL=0
MOVL C01647 V=800.0 PL=0
MOVL C01648 V=800.0 PL=0
MOVL C01649 V=800.0 PL=0
MOVL C01650 V=800.0 PL=0
MOVL C01651 V=800.0 PL=0
MOVL C01652 V=800.0 PL=0
MOVL C01653 V=800.0 PL=0
MOVL C01654 V=800.0 PL=0
MOVL C01655 V=800.0 PL=0
MOVL C01656 V=800.0 PL=0
MOVL C01657 V=800.0 PL=0
MOVL C01658 V=800.0 PL=0
MOVL C01659 V=800.0 PL=0
MOVL C01660 V=800.0 PL=0
MOVL C01661 V=800.0 PL=0
MOVL C01662 V=800.0 PL=0
MOVL C01663 V=800.0 PL=0
MOVL C01664 V=800.0 PL=0
MOVL C01665 V=800.0 PL=0
MOVL C01666 V=800.0 PL=0
MOVL C01667 V=800.0 PL=0
MOVL C01668 V=800.0 PL=0
MOVL C01669 V=800.0 PL=0
MOVL C01670 V=800.0 PL=0
MOVL C01671 V=800.0 PL=0
MOVL C01672 V=800.0 PL=0
MOVL C01673 V=800.0 PL=0
MOVL C01674 V=800.0 PL=0
MOVL C01675 V=800.0 PL=0
MOVL C01676 V=800.0 PL=0
MOVL C01677 V=800.0 PL=0
MOVL C01678 V=800.0 PL=0
MOVL C01679 V=800.0 PL=0
MOVL C01680 V=800.0 PL=0
MOVL C01681 V=800.0 PL=0
MOVL C01682 V=800.0 PL=0
MOVL C01683 V=800.0 PL=0
MOVL C01684 V=800.0 PL=0
MOVL C01685 V=800.0 PL=0
MOVL C01686 V=800.0 PL=0
MOVL C01687 V=800.0 PL=0
MOVL C01688 V=800.0 PL=0
MOVL C01689 V=800.0 PL=0
MOVL C01690 V=800.0 PL=0
MOVL C01691 V=800.0 PL=0
MOVL C01692 V=800.0 PL=0
MOVL C01693 V=800.0 PL=0
MOVL C01694 V=800.0 PL=0
MOVL C01695 V=800.0 PL=0
MOVL C01696 V=800.0 PL=0
MOVL C01697 V=800.0 PL=0
MOVL C01698 V=800.0 PL=0
MOVL C01699 V=800.0 PL=0
MOVL C01700 V=800.0 PL=0
MOVL C01701 V=800.0 PL=0
MOVL C01702 V=800.0 PL=0
MOVL C01703 V=800.0 PL=0
MOVL C01704 V=800.0 PL=0
MOVL C01705 V=800.0 PL=0
MOVL C01706 V=800.0 PL=0
MOVL C01707 V=800.0 PL=0
MOVL C01708 V=800.0 PL=0
MOVL C01709 V=800.0 PL=0
MOVL C01710 V=800.0 PL=0
MOVL C01711 V=800.0 PL=0
MOVL C01712 V=800.0 PL=0
MOVL C01713 V=800.0 PL=0
MOVL C01714 V=800.0 PL=0
MOVL C01715 V=800.0 PL=0
MOVL C01716 V=800.0 PL=0
MOVL C01717 V=800.0 PL=0
MOVL C01718 V=800.0 PL=0
MOVL C01719 V=800.0 PL=0
MOVL C01720 V=800.0 PL=0
MOVL C01721 V=800.0 PL=0
MOVL C01722 V=800.0 PL=0
MOVL C01723 V=800.0 PL=0
MOVL C01724 V=800.0 PL=0
MOVL C01725 V=800.0 PL=0
MOVL C01726 V=800.0 PL=0
MOVL C01727 V=800.0 PL=0
MOVL C01728 V=800.0 PL=0
MOVL C01729 V=800.0 PL=0
MOVL C01730 V=800.0 PL=0
MOVL C01731 V=800.0 PL=0
MOVL C01732 V=800.0 PL=0
MOVL C01733 V=800.0 PL=0
MOVL C01734 V=800.0 PL=0
MOVL C01735 V=800.0 PL=0
MOVL C01736 V=800.0 PL=0
MOVL C01737 V=800.0 PL=0
MOVL C01738 V=800.0 PL=0
MOVL C01739 V=800.0 PL=0
MOVL C01740 V=800.0 PL=0
MOVL C01741 V=800.0 PL=0
MOVL C01742 V=800.0 PL=0
MOVL C01743 V=800.0 PL=0
MOVL C01744 V=800.0 PL=0
MOVL C01745 V=800.0 PL=0
MOVL C01746 V=800.0 PL=0
MOVL C01747 V=800.0 PL=0
MOVL C01748 V=800.0 PL=0
MOVL C01749 V=800.0 PL=0
MOVL C01750 V=800.0 PL=0
MOVL C01751 V=800.0 PL=0
MOVL C01752 V=800.0 PL=0
MOVL C01753 V=800.0 PL=0
MOVL C01754 V=800.0 PL=0
MOVL C01755 V=800.0 PL=0
MOVL C01756 V=800.0 PL=0
MOVL C01757 V=800.0 PL=0
MOVL C01758 V=800.0 PL=0
MOVL C01759 V=800.0 PL=0
MOVL C01760 V=800.0 PL=0
MOVL C01761 V=800.0 PL=0
MOVL C01762 V=800.0 PL=0
MOVL C01763 V=800.0 PL=0
MOVL C01764 V=800.0 PL=0
MOVL C01765 V=800.0 PL=0
MOVL C01766 V=800.0 PL=0
MOVL C01767 V=800.0 PL=0
MOVL C01768 V=800.0 PL=0
MOVL C01769 V=800.0 PL=0
MOVL C01770 V=800.0 PL=0
MOVL C01771 V=800.0 PL=0
MOVL C01772 V=800.0 PL=0
MOVL C01773 V=800.0 PL=0
MOVL C01774 V=800.0 PL=0
MOVL C01775 V=800.0 PL=0
MOVL C01776 V=800.0 PL=0
MOVL C01777 V=800.0 PL=0
MOVL C01778 V=800.0 PL=0
MOVL C01779 V=800.0 PL=0
MOVL C01780 V=800.0 PL=0
MOVL C01781 V=800.0 PL=0
MOVL C01782 V=800.0 PL=0
MOVL C01783 V=800.0 PL=0
MOVL C01784 V=800.0 PL=0
MOVL C01785 V=800.0 PL=0
MOVL C01786 V=800.0 PL=0
MOVL C01787 V=800.0 PL=0
MOVL C01788 V=800.0 PL=0
MOVL C01789 V=800.0 PL=0
MOVL C01790 V=800.0 PL=0
MOVL C01791 V=800.0 PL=0
MOVL C01792 V=800.0 PL=0
MOVL C01793 V=800.0 PL=0
MOVL C01794 V=800.0 PL=0
MOVL C01795 V=800.0 PL=0
MOVL C01796 V=800.0 PL=0
MOVL C01797 V=800.0 PL=0
MOVL C01798 V=800.0 PL=0
MOVL C01799 V=800.0 PL=0
MOVL C01800 V=800.0 PL=0
MOVL C01801 V=800.0 PL=0
MOVL C01802 V=800.0 PL=0
MOVL C01803 V=800.0 PL=0
MOVL C01804 V=800.0 PL=0
MOVL C01805 V=800.0 PL=0
MOVL C01806 V=800.0 PL=0
MOVL C01807 V=800.0 PL=0
MOVL C01808 V=800.0 PL=0
MOVL C01809 V=800.0 PL=0
MOVL C01810 V=800.0 PL=0
MOVL C01811 V=800.0 PL=0
MOVL C01812 V=800.0 PL=0
MOVL C01813 V=800.0 PL=0
MOVL C01814 V=800.0 PL=0
MOVL C01815 V=800.0 PL=0
MOVL C01816 V=800.0 PL=0
MOVL C01817 V=800.0 PL=0
MOVL C01818 V=800.0 PL=0
MOVL C01819 V=800.0 PL=0
MOVL C01820 V=800.0 PL=0
MOVL C01821 V=800.0 PL=0
MOVL C01822 V=800.0 PL=0
MOVL C01823 V=800.0 PL=0
MOVL C01824 V=800.0 PL=0
MOVL C01825 V=800.0 PL=0
MOVL C01826 V=800.0 PL=0
MOVL C01827 V=800.0 PL=0
MOVL C01828 V=800.0 PL=0
MOVL C01829 V=800.0 PL=0
MOVL C01830 V=800.0 PL=0
MOVL C01831 V=800.0 PL=0
MOVL C01832 V=800.0 PL=0
MOVL C01833 V=800.0 PL=0
MOVL C01834 V=800.0 PL=0
MOVL C01835 V=800.0 PL=0
MOVL C01836 V=800.0 PL=0
MOVL C01837 V=800.0 PL=0
MOVL C01838 V=800.0 PL=0
MOVL C01839 V=800.0 PL=0
MOVL C01840 V=800.0 PL=0
MOVL C01841 V=800.0 PL=0
MOVL C01842 V=800.0 PL=0
MOVL C01843 V=800.0 PL=0
MOVL C01844 V=800.0 PL=0
MOVL C01845 V=800.0 PL=0
MOVL C01846 V=800.0 PL=0
MOVL C01847 V=800.0 PL=0
MOVL C01848 V=800.0 PL=0
MOVL C01849 V=800.0 PL=0
MOVL C01850 V=800.0 PL=0
MOVL C01851 V=800.0 PL=0
MOVL C01852 V=800.0 PL=0
MOVL C01853 V=800.0 PL=0
MOVL C01854 V=800.0 PL=0
MOVL C01855 V=800.0 PL=0
MOVL C01856 V=800.0 PL=0
MOVL C01857 V=800.0 PL=0
MOVL C01858 V=800.0 PL=0
MOVL C01859 V=800.0 PL=0
MOVL C01860 V=800.0 PL=0
MOVL C01861 V=800.0 PL=0
MOVL C01862 V=800.0 PL=0
MOVL C01863 V=800.0 PL=0
MOVL C01864 V=800.0 PL=0
MOVL C01865 V=800.0 PL=0
MOVL C01866 V=800.0 PL=0
MOVL C01867 V=800.0 PL=0
MOVL C01868 V=800.0 PL=0
MOVL C01869 V=800.0 PL=0
MOVL C01870 V=800.0 PL=0
MOVL C01871 V=800.0 PL=0
MOVL C01872 V=800.0 PL=0
MOVL C01873 V=800.0 PL=0
MOVL C01874 V=800.0 PL=0
MOVL C01875 V=800.0 PL=0
MOVL C01876 V=800.0 PL=0
MOVL C01877 V=800.0 PL=0
MOVL C01878 V=800.0 PL=0
MOVL C01879 V=800.0 PL=0
MOVL C01880 V=800.0 PL=0
MOVL C01881 V=800.0 PL=0
MOVL C01882 V=800.0 PL=0
MOVL C01883 V=800.0 PL=0
MOVL C01884 V=800.0 PL=0
MOVL C01885 V=800.0 PL=0
MOVL C01886 V=800.0 PL=0
MOVL C01887 V=800.0 PL=0
MOVL C01888 V=800.0 PL=0
MOVL C01889 V=800.0 PL=0
MOVL C01890 V=800.0 PL=0
MOVL C01891 V=800.0 PL=0
MOVL C01892 V=800.0 PL=0
MOVL C01893 V=800.0 PL=0
MOVL C01894 V=800.0 PL=0
MOVL C01895 V=800.0 PL=0
MOVL C01896 V=800.0 PL=0
MOVL C01897 V=800.0 PL=0
MOVL C01898 V=800.0 PL=0
MOVL C01899 V=800.0 PL=0
MOVL C01900 V=800.0 PL=0
MOVL C01901 V=800.0 PL=0
MOVL C01902 V=800.0 PL=0
MOVL C01903 V=800.0 PL=0
MOVL C01904 V=800.0 PL=0
MOVL C01905 V=800.0 PL=0
MOVL C01906 V=800.0 PL=0
MOVL C01907 V=800.0 PL=0
MOVL C01908 V=800.0 PL=0
MOVL C01909 V=800.0 PL=0
MOVL C01910 V=800.0 PL=0
MOVL C01911 V=800.0 PL=0
MOVL C01912 V=800.0 PL=0
MOVL C01913 V=800.0 PL=0
MOVL C01914 V=800.0 PL=0
MOVL C01915 V=800.0 PL=0
MOVL C01916 V=800.0 PL=0
MOVL C01917 V=800.0 PL=0
MOVL C01918 V=800.0 PL=0
MOVL C01919 V=800.0 PL=0
MOVL C01920 V=800.0 PL=0
MOVL C01921 V=800.0 PL=0
MOVL C01922 V=800.0 PL=0
MOVL C01923 V=800.0 PL=0
MOVL C01924 V=800.0 PL=0
MOVL C01925 V=800.0 PL=0
MOVL C01926 V=800.0 PL=0
MOVL C01927 V=800.0 PL=0
MOVL C01928 V=800.0 PL=0
MOVL C01929 V=800.0 PL=0
MOVL C01930 V=800.0 PL=0
MOVL C01931 V=800.0 PL=0
MOVL C01932 V=800.0 PL=0
MOVL C01933 V=800.0 PL=0
MOVL C01934 V=800.0 PL=0
MOVL C01935 V=800.0 PL=0
MOVL C01936 V=800.0 PL=0
MOVL C01937 V=800.0 PL=0
MOVL C01938 V=800.0 PL=0
MOVL C01939 V=800.0 PL=0
MOVL C01940 V=800.0 PL=0
MOVL C01941 V=800.0 PL=0
MOVL C01942 V=800.0 PL=0
MOVL C01943 V=800.0 PL=0
MOVL C01944 V=800.0 PL=0
MOVL C01945 V=800.0 PL=0
MOVL C01946 V=800.0 PL=0
MOVL C01947 V=800.0 PL=0
MOVL C01948 V=800.0 PL=0
MOVL C01949 V=800.0 PL=0
MOVL C01950 V=800.0 PL=0
MOVL C01951 V=800.0 PL=0
MOVL C01952 V=800.0 PL=0
MOVL C01953 V=800.0 PL=0
MOVL C01954 V=800.0 PL=0
MOVL C01955 V=800.0 PL=0
MOVL C01956 V=800.0 PL=0
MOVL C01957 V=800.0 PL=0
MOVL C01958 V=800.0 PL=0
MOVL C01959 V=800.0 PL=0
MOVL C01960 V=800.0 PL=0
MOVL C01961 V=800.0 PL=0
MOVL C01962 V=800.0 PL=0
MOVL C01963 V=800.0 PL=0
MOVL C01964 V=800.0 PL=0
MOVL C01965 V=800.0 PL=0
MOVL C01966 V=800.0 PL=0
MOVL C01967 V=800.0 PL=0
MOVL C01968 V=800.0 PL=0
MOVL C01969 V=800.0 PL=0
MOVL C01970 V=800.0 PL=0
MOVL C01971 V=800.0 PL=0
MOVL C01972 V=800.0 PL=0
MOVL C01973 V=800.0 PL=0
MOVL C01974 V=800.0 PL=0
MOVL C01975 V=800.0 PL=0
MOVL C01976 V=800.0 PL=0
MOVL C01977 V=800.0 PL=0
MOVL C01978 V=800.0 PL=0
MOVL C01979 V=800.0 PL=0
MOVL C01980 V=800.0 PL=0
MOVL C01981 V=800.0 PL=0
MOVL C01982 V=800.0 PL=0
MOVL C01983 V=800.0 PL=0
MOVL C01984 V=800.0 PL=0
MOVL C01985 V=800.0 PL=0
MOVL C01986 V=800.0 PL=0
MOVL C01987 V=800.0 PL=0
MOVL C01988 V=800.0 PL=0
MOVL C01989 V=800.0 PL=0
MOVL C01990 V=800.0 PL=0
MOVL C01991 V=800.0 PL=0
MOVL C01992 V=800.0 PL=0
MOVL C01993 V=800.0 PL=0
MOVL C01994 V=800.0 PL=0
MOVL C01995 V=800.0 PL=0
MOVL C01996 V=800.0 PL=0
MOVL C01997 V=800.0 PL=0
MOVL C01998 V=800.0 PL=0
MOVL C01999 V=800.0 PL=0
MOVL C02000 V=800.0 PL=0
MOVL C02001 V=800.0 PL=0
MOVL C02002 V=800.0 PL=0
MOVL C02003 V=800.0 PL=0
MOVL C02004 V=800.0 PL=0
MOVL C02005 V=800.0 PL=0
MOVL C02006 V=800.0 PL=0
MOVL C02007 V=800.0 PL=0
MOVL C02008 V=800.0 PL=0
MOVL C02009 V=800.0 PL=0
MOVL C02010 V=800.0 PL=0
MOVL C02011 V=800.0 PL=0
MOVL C02012 V=800.0 PL=0
MOVL C02013 V=800.0 PL=0
MOVL C02014 V=800.0 PL=0
MOVL C02015 V=800.0 PL=0
MOVL C02016 V=800.0 PL=0
MOVL C02017 V=800.0 PL=0
MOVL C02018 V=800.0 PL=0
MOVL C02019 V=800.0 PL=0
MOVL C02020 V=800.0 PL=0
MOVL C02021 V=800.0 PL=0
MOVL C02022 V=800.0 PL=0
MOVL C02023 V=800.0 PL=0
MOVL C02024 V=800.0 PL=0
MOVL C02025 V=800.0 PL=0
MOVL C02026 V=800.0 PL=0
MOVL C02027 V=800.0 PL=0
MOVL C02028 V=800.0 PL=0
MOVL C02029 V=800.0 PL=0
MOVL C02030 V=800.0 PL=0
MOVL C02031 V=800.0 PL=0
